LIN {X 0,Y 340.688,Z 497.175,A -85,B 0,C 180,E1 -14276.154,E2 -14276.154} C_VEL
LIN {X 0,Y 340.77,Z 497.165,A -85,B 0,C 180,E1 -14280.333,E2 -14280.333} C_VEL
LIN {X 0,Y 340.804,Z 497.363,A -85,B 0,C 180,E1 -14283.682,E2 -14283.682} C_VEL
LIN {X 0,Y 341.004,Z 498.318,A -85,B 0,C 180,E1 -14283.975,E2 -14283.975} C_VEL
LIN {X 0,Y 342.467,Z 500.978,A -85,B 0,C 180,E1 -14284.442,E2 -14284.442} C_VEL
LIN {X 0,Y 344.948,Z 503.079,A -85,B 0,C 180,E1 -14285.106,E2 -14285.106} C_VEL
LIN {X 0,Y 346.96,Z 506.236,A -85,B 0,C 180,E1 -14285.714,E2 -14285.714} C_VEL
LIN {X 0,Y 349.668,Z 508.622,A -85,B 0,C 180,E1 -14286.488,E2 -14286.488} C_VEL
LIN {X 0,Y 352.115,Z 512,A -85,B 0,C 180,E1 -14287.255,E2 -14287.255} C_VEL
LIN {X 0,Y 355.034,Z 514.578,A -85,B 0,C 180,E1 -14288.144,E2 -14288.144} C_VEL
LIN {X 0,Y 357.879,Z 518.099,A -85,B 0,C 180,E1 -14289.088,E2 -14289.088} C_VEL
LIN {X 0,Y 360.863,Z 520.59,A -85,B 0,C 180,E1 -14290.074,E2 -14290.074} C_VEL
LIN {X 0,Y 363.526,Z 523.831,A -85,B 0,C 180,E1 -14291.039,E2 -14291.039} C_VEL
LIN {X 0,Y 367.234,Z 526.893,A -85,B 0,C 180,E1 -14292.394,E2 -14292.394} C_VEL
LIN {X 0,Y 369.963,Z 530.151,A -85,B 0,C 180,E1 -14293.522,E2 -14293.522} C_VEL
LIN {X 0,Y 373.28,Z 532.615,A -85,B 0,C 180,E1 -14294.922,E2 -14294.922} C_VEL
LIN {X 0,Y 374.392,Z 533.739,A -85,B 0,C 180,E1 -14295.436,E2 -14295.436} C_VEL
LIN {X 0,Y 377.136,Z 536.901,A -85,B 0,C 180,E1 -14296.811,E2 -14296.811} C_VEL
LIN {X 0,Y 380.19,Z 539.057,A -85,B 0,C 180,E1 -14298.441,E2 -14298.441} C_VEL
LIN {X 0,Y 381.738,Z 539.964,A -85,B 0,C 180,E1 -14299.348,E2 -14299.348} C_VEL
LIN {X 0,Y 384.051,Z 542.876,A -85,B 0,C 180,E1 -14301.001,E2 -14301.001} C_VEL
LIN {X 0,Y 386.257,Z 544.769,A -85,B 0,C 180,E1 -14302.826,E2 -14302.826} C_VEL
LIN {X 0,Y 388.334,Z 545.981,A -85,B 0,C 180,E1 -14305.057,E2 -14305.057} C_VEL
LIN {X 0,Y 389.706,Z 546.532,A -85,B 0,C 180,E1 -14307.322,E2 -14307.322} C_VEL
LIN {X 0,Y 390.171,Z 546.851,A -85,B 0,C 180,E1 -14308.968,E2 -14308.968} C_VEL
LIN {X 0,Y 390.171,Z 546.854,A -85,B 0,C 180,E1 -14311.032,E2 -14311.032} C_VEL
LIN {X 0,Y 389.505,Z 546.374,A -85,B 0,C 180,E1 -14313.103,E2 -14313.103} C_VEL
LIN {X 0,Y 388.131,Z 545.895,A -85,B 0,C 180,E1 -14315.197,E2 -14315.197} C_VEL
LIN {X 0,Y 386.111,Z 544.648,A -85,B 0,C 180,E1 -14317.32,E2 -14317.32} C_VEL
LIN {X 0,Y 384.057,Z 542.843,A -85,B 0,C 180,E1 -14318.997,E2 -14318.997} C_VEL
LIN {X 0,Y 381.688,Z 539.897,A -85,B 0,C 180,E1 -14320.684,E2 -14320.684} C_VEL
LIN {X 0,Y 378.266,Z 537.815,A -85,B 0,C 180,E1 -14322.602,E2 -14322.602} C_VEL
LIN {X 0,Y 375.358,Z 535.009,A -85,B 0,C 180,E1 -14324.087,E2 -14324.087} C_VEL
LIN {X 0,Y 373.457,Z 532.737,A -85,B 0,C 180,E1 -14325.002,E2 -14325.002} C_VEL
LIN {X 0,Y 369.922,Z 530.118,A -85,B 0,C 180,E1 -14326.495,E2 -14326.495} C_VEL
LIN {X 0,Y 366.356,Z 526.09,A -85,B 0,C 180,E1 -14327.934,E2 -14327.934} C_VEL
LIN {X 0,Y 362.932,Z 523.255,A -85,B 0,C 180,E1 -14329.176,E2 -14329.176} C_VEL
LIN {X 0,Y 360.249,Z 519.926,A -85,B 0,C 180,E1 -14330.142,E2 -14330.142} C_VEL
LIN {X 0,Y 357.091,Z 517.292,A -85,B 0,C 180,E1 -14331.176,E2 -14331.176} C_VEL
LIN {X 0,Y 354.349,Z 513.844,A -85,B 0,C 180,E1 -14332.076,E2 -14332.076} C_VEL
LIN {X 0,Y 351.341,Z 511.117,A -85,B 0,C 180,E1 -14332.986,E2 -14332.986} C_VEL
LIN {X 0,Y 349.194,Z 508.114,A -85,B 0,C 180,E1 -14333.651,E2 -14333.651} C_VEL
LIN {X 0,Y 346.5,Z 505.693,A -85,B 0,C 180,E1 -14334.417,E2 -14334.417} C_VEL
LIN {X 0,Y 344.728,Z 502.722,A -85,B 0,C 180,E1 -14334.962,E2 -14334.962} C_VEL
LIN {X 0,Y 342.3,Z 500.782,A -85,B 0,C 180,E1 -14335.604,E2 -14335.604} C_VEL
LIN {X 0,Y 340.899,Z 497.904,A -85,B 0,C 180,E1 -14336.105,E2 -14336.105} C_VEL
LIN {X 0,Y 340.809,Z 497.209,A -85,B 0,C 180,E1 -14336.483,E2 -14336.483} C_VEL
LIN {X 0,Y 340.758,Z 497.166,A -85,B 0,C 180,E1 -14339.978,E2 -14339.978} C_VEL
LIN {X 0,Y 340.688,Z 497.175,A -85,B 0,C 180,E1 -14343.846,E2 -14343.846} C_VEL
LIN {X 0,Y 340.7,Z 497.141,A -85,B 0,C 180,E1 -14346.741,E2 -14346.741} C_VEL
LIN {X 0,Y 340.758,Z 497.161,A -85,B 0,C 180,E1 -14350.262,E2 -14350.262} C_VEL
LIN {X 0,Y 340.772,Z 497.12,A -85,B 0,C 180,E1 -14353.795,E2 -14353.795} C_VEL
LIN {X 0,Y 340.755,Z 497.164,A -85,B 0,C 180,E1 -14357.109,E2 -14357.109} C_VEL
LIN {X 0,Y 340.727,Z 497.161,A -85,B 0,C 180,E1 -14360.252,E2 -14360.252} C_VEL
LIN {X 0,Y 340.703,Z 497.158,A -85,B 0,C 180,E1 -14363.559,E2 -14363.559} C_VEL
LIN {X 0,Y 340.688,Z 497.172,A -85,B 0,C 180,E1 -14366.154,E2 -14366.154} C_VEL
LIN {X 0,Y 340.768,Z 497.147,A -85,B 0,C 180,E1 -14370.333,E2 -14370.333} C_VEL
LIN {X 0,Y 340.797,Z 497.156,A -85,B 0,C 180,E1 -14373.02,E2 -14373.02} C_VEL
LIN {X 0,Y 340.753,Z 497.147,A -85,B 0,C 180,E1 -14374.696,E2 -14374.696} C_VEL
LIN {X 0,Y 340.07,Z 497.23,A -85,B 0,C 180,E1 -14375.683,E2 -14375.683} C_VEL
LIN {X 0,Y 337.176,Z 497.602,A -85,B 0,C 180,E1 -14377.288,E2 -14377.288} C_VEL
LIN {X 0,Y 334.755,Z 497.913,A -85,B 0,C 180,E1 -14378.587,E2 -14378.587} C_VEL
LIN {X 0,Y 333.756,Z 498.034,A -85,B 0,C 180,E1 -14379.594,E2 -14379.594} C_VEL
LIN {X 0,Y 333.696,Z 498.037,A -85,B 0,C 180,E1 -14379.935,E2 -14379.935} C_VEL
LIN {X 0,Y 333.738,Z 498.014,A -85,B 0,C 180,E1 -14382.854,E2 -14382.854} C_VEL
LIN {X 0,Y 333.789,Z 498.032,A -85,B 0,C 180,E1 -14386.609,E2 -14386.609} C_VEL
LIN {X 0,Y 333.843,Z 497.997,A -85,B 0,C 180,E1 -14390.305,E2 -14390.305} C_VEL
LIN {X 0,Y 334,Z 498,A -85,B 0,C 180,E1 -14392.748,E2 -14392.748} C_VEL
LIN {X 0,Y 333.807,Z 498.022,A -85,B 0,C 180,E1 -14395.17,E2 -14395.17} C_VEL
LIN {X 0,Y 334.1,Z 497.963,A -85,B 0,C 180,E1 -14397.589,E2 -14397.589} C_VEL
LIN {X 0,Y 334.239,Z 497.962,A -85,B 0,C 180,E1 -14400.001,E2 -14400.001} C_VEL
LIN {X 0,Y 334.1,Z 497.991,A -85,B 0,C 180,E1 -14402.412,E2 -14402.412} C_VEL
LIN {X 0,Y 334.009,Z 497.974,A -85,B 0,C 180,E1 -14406.04,E2 -14406.04} C_VEL
LIN {X 0,Y 333.978,Z 498.003,A -85,B 0,C 180,E1 -14408.502,E2 -14408.502} C_VEL
LIN {X 0,Y 333.784,Z 498.014,A -85,B 0,C 180,E1 -14412.155,E2 -14412.155} C_VEL
LIN {X 0,Y 333.771,Z 498.027,A -85,B 0,C 180,E1 -14415.887,E2 -14415.887} C_VEL
LIN {X 0,Y 333.79,Z 498.023,A -85,B 0,C 180,E1 -14418.656,E2 -14418.656} C_VEL
LIN {X 0,Y 333.651,Z 498.037,A -85,B 0,C 180,E1 -14422.282,E2 -14422.282} C_VEL
LIN {X 0,Y 333.729,Z 498.024,A -85,B 0,C 180,E1 -14426.247,E2 -14426.247} C_VEL
LIN {X 0,Y 333.685,Z 498.039,A -85,B 0,C 180,E1 -14428.975,E2 -14428.975} C_VEL
LIN {X 0,Y 333.639,Z 498.035,A -85,B 0,C 180,E1 -14432.588,E2 -14432.588} C_VEL
LIN {X 0,Y 333.673,Z 498.047,A -85,B 0,C 180,E1 -14436.14,E2 -14436.14} C_VEL
LIN {X 0,Y 333.669,Z 498.045,A -85,B 0,C 180,E1 -14439.19,E2 -14439.19} C_VEL
LIN {X 0,Y 333.663,Z 498.041,A -85,B 0,C 180,E1 -14442.507,E2 -14442.507} C_VEL
LIN {X 0,Y 333.595,Z 498.033,A -85,B 0,C 180,E1 -14445.956,E2 -14445.956} C_VEL
LIN {X 0,Y 333.646,Z 498.051,A -85,B 0,C 180,E1 -14449.316,E2 -14449.316} C_VEL
LIN {X 0,Y 333.679,Z 498.02,A -85,B 0,C 180,E1 -14453.317,E2 -14453.317} C_VEL
LIN {X 0,Y 333.95,Z 499.209,A -85,B 0,C 180,E1 -14453.896,E2 -14453.896} C_VEL
LIN {X 0,Y 336.328,Z 509.72,A -85,B 0,C 180,E1 -14457.448,E2 -14457.448} C_VEL
LIN {X 0,Y 338.327,Z 519.735,A -85,B 0,C 180,E1 -14460.699,E2 -14460.699} C_VEL
LIN {X 0,Y 340.345,Z 524.973,A -85,B 0,C 180,E1 -14461.07,E2 -14461.07} C_VEL
LIN {X 0,Y 342.174,Z 531.358,A -85,B 0,C 180,E1 -14461.387,E2 -14461.387} C_VEL
LIN {X 0,Y 347.112,Z 554.272,A -85,B 0,C 180,E1 -14462.352,E2 -14462.352} C_VEL
LIN {X 0,Y 349.193,Z 565.536,A -85,B 0,C 180,E1 -14462.784,E2 -14462.784} C_VEL
LIN {X 0,Y 346.958,Z 654.163,A -85,B 0,C 180,E1 -14464.626,E2 -14464.626} C_VEL
LIN {X 0,Y 346.331,Z 665.498,A -85,B 0,C 180,E1 -14464.978,E2 -14464.978} C_VEL
LIN {X 0,Y 345.507,Z 676.04,A -85,B 0,C 180,E1 -14465.436,E2 -14465.436} C_VEL
LIN {X 0,Y 344.42,Z 687.192,A -85,B 0,C 180,E1 -14466.075,E2 -14466.075} C_VEL
LIN {X 0,Y 343.36,Z 697.164,A -85,B 0,C 180,E1 -14466.796,E2 -14466.796} C_VEL
LIN {X 0,Y 342.068,Z 706.938,A -85,B 0,C 180,E1 -14467.645,E2 -14467.645} C_VEL
LIN {X 0,Y 340.804,Z 716.811,A -85,B 0,C 180,E1 -14468.688,E2 -14468.688} C_VEL
LIN {X 0,Y 339.314,Z 726.229,A -85,B 0,C 180,E1 -14469.859,E2 -14469.859} C_VEL
LIN {X 0,Y 338.152,Z 733.431,A -85,B 0,C 180,E1 -14470.893,E2 -14470.893} C_VEL
LIN {X 0,Y 336.765,Z 742.226,A -85,B 0,C 180,E1 -14472.386,E2 -14472.386} C_VEL
LIN {X 0,Y 335.551,Z 749.751,A -85,B 0,C 180,E1 -14473.888,E2 -14473.888} C_VEL
LIN {X 0,Y 334.658,Z 756.23,A -85,B 0,C 180,E1 -14475.404,E2 -14475.404} C_VEL
LIN {X 0,Y 333.703,Z 762.773,A -85,B 0,C 180,E1 -14477.225,E2 -14477.225} C_VEL
LIN {X 0,Y 332.883,Z 768.204,A -85,B 0,C 180,E1 -14479.047,E2 -14479.047} C_VEL
LIN {X 0,Y 332.439,Z 772.651,A -85,B 0,C 180,E1 -14480.877,E2 -14480.877} C_VEL
LIN {X 0,Y 332.172,Z 776.198,A -85,B 0,C 180,E1 -14482.707,E2 -14482.707} C_VEL
LIN {X 0,Y 332.004,Z 778.556,A -85,B 0,C 180,E1 -14484.224,E2 -14484.224} C_VEL
LIN {X 0,Y 331.962,Z 780.825,A -85,B 0,C 180,E1 -14486.359,E2 -14486.359} C_VEL
LIN {X 0,Y 331.922,Z 782.114,A -85,B 0,C 180,E1 -14488.787,E2 -14488.787} C_VEL
LIN {X 0,Y 331.969,Z 782.367,A -85,B 0,C 180,E1 -14490,E2 -14490} C_VEL
LIN {X 0,Y 331.913,Z 781.641,A -85,B 0,C 180,E1 -14492.427,E2 -14492.427} C_VEL
LIN {X 0,Y 331.962,Z 780.824,A -85,B 0,C 180,E1 -14493.641,E2 -14493.641} C_VEL
LIN {X 0,Y 332.044,Z 778.139,A -85,B 0,C 180,E1 -14496.075,E2 -14496.075} C_VEL
LIN {X 0,Y 332.241,Z 775.182,A -85,B 0,C 180,E1 -14497.903,E2 -14497.903} C_VEL
LIN {X 0,Y 332.572,Z 771.353,A -85,B 0,C 180,E1 -14499.733,E2 -14499.733} C_VEL
LIN {X 0,Y 333.149,Z 766.589,A -85,B 0,C 180,E1 -14501.561,E2 -14501.561} C_VEL
LIN {X 0,Y 334.095,Z 759.643,A -85,B 0,C 180,E1 -14503.689,E2 -14503.689} C_VEL
LIN {X 0,Y 335.126,Z 752.272,A -85,B 0,C 180,E1 -14505.544,E2 -14505.544} C_VEL
LIN {X 0,Y 336.23,Z 745.35,A -85,B 0,C 180,E1 -14507.015,E2 -14507.015} C_VEL
LIN {X 0,Y 337.581,Z 737.069,A -85,B 0,C 180,E1 -14508.51,E2 -14508.51} C_VEL
LIN {X 0,Y 338.972,Z 728.348,A -85,B 0,C 180,E1 -14509.846,E2 -14509.846} C_VEL
LIN {X 0,Y 340.426,Z 719.291,A -85,B 0,C 180,E1 -14511.02,E2 -14511.02} C_VEL
LIN {X 0,Y 341.744,Z 710.224,A -85,B 0,C 180,E1 -14512.02,E2 -14512.02} C_VEL
LIN {X 0,Y 342.927,Z 700.672,A -85,B 0,C 180,E1 -14512.916,E2 -14512.916} C_VEL
LIN {X 0,Y 344.092,Z 690.413,A -85,B 0,C 180,E1 -14513.71,E2 -14513.71} C_VEL
LIN {X 0,Y 345.127,Z 680.119,A -85,B 0,C 180,E1 -14514.353,E2 -14514.353} C_VEL
LIN {X 0,Y 346.156,Z 668.235,A -85,B 0,C 180,E1 -14514.915,E2 -14514.915} C_VEL
LIN {X 0,Y 346.807,Z 656.819,A -85,B 0,C 180,E1 -14515.306,E2 -14515.306} C_VEL
LIN {X 0,Y 347.758,Z 626.709,A -85,B 0,C 180,E1 -14515.954,E2 -14515.954} C_VEL
LIN {X 0,Y 349.181,Z 565.129,A -85,B 0,C 180,E1 -14517.226,E2 -14517.226} C_VEL
LIN {X 0,Y 344.511,Z 541.355,A -85,B 0,C 180,E1 -14518.171,E2 -14518.171} C_VEL
LIN {X 0,Y 340.705,Z 525.852,A -85,B 0,C 180,E1 -14518.876,E2 -14518.876} C_VEL
LIN {X 0,Y 338.363,Z 519.983,A -85,B 0,C 180,E1 -14519.265,E2 -14519.265} C_VEL
LIN {X 0,Y 337.891,Z 517.596,A -85,B 0,C 180,E1 -14519.946,E2 -14519.946} C_VEL
LIN {X 0,Y 336.034,Z 508.584,A -85,B 0,C 180,E1 -14522.94,E2 -14522.94} C_VEL
LIN {X 0,Y 333.955,Z 499.268,A -85,B 0,C 180,E1 -14526.103,E2 -14526.103} C_VEL
LIN {X 0,Y 333.679,Z 498.035,A -85,B 0,C 180,E1 -14526.683,E2 -14526.683} C_VEL
LIN {X 0,Y 333.646,Z 498.051,A -85,B 0,C 180,E1 -14530.684,E2 -14530.684} C_VEL
LIN {X 0,Y 333.592,Z 498.034,A -85,B 0,C 180,E1 -14534.25,E2 -14534.25} C_VEL
LIN {X 0,Y 333.671,Z 498.038,A -85,B 0,C 180,E1 -14537.622,E2 -14537.622} C_VEL
LIN {X 0,Y 333.674,Z 498.038,A -85,B 0,C 180,E1 -14541.196,E2 -14541.196} C_VEL
LIN {X 0,Y 333.682,Z 498.041,A -85,B 0,C 180,E1 -14545.225,E2 -14545.225} C_VEL
LIN {X 0,Y 333.627,Z 498.046,A -85,B 0,C 180,E1 -14548.221,E2 -14548.221} C_VEL
LIN {X 0,Y 333.685,Z 498.039,A -85,B 0,C 180,E1 -14551.025,E2 -14551.025} C_VEL
LIN {X 0,Y 333.729,Z 498.024,A -85,B 0,C 180,E1 -14553.753,E2 -14553.753} C_VEL
LIN {X 0,Y 333.651,Z 498.037,A -85,B 0,C 180,E1 -14557.718,E2 -14557.718} C_VEL
LIN {X 0,Y 333.788,Z 498.026,A -85,B 0,C 180,E1 -14561.589,E2 -14561.589} C_VEL
LIN {X 0,Y 333.802,Z 498.006,A -85,B 0,C 180,E1 -14565.576,E2 -14565.576} C_VEL
LIN {X 0,Y 333.827,Z 498.021,A -85,B 0,C 180,E1 -14569.077,E2 -14569.077} C_VEL
LIN {X 0,Y 334.007,Z 497.988,A -85,B 0,C 180,E1 -14572.747,E2 -14572.747} C_VEL
LIN {X 0,Y 333.803,Z 498.003,A -85,B 0,C 180,E1 -14575.168,E2 -14575.168} C_VEL
LIN {X 0,Y 334.1,Z 497.991,A -85,B 0,C 180,E1 -14577.588,E2 -14577.588} C_VEL
LIN {X 0,Y 334.239,Z 497.962,A -85,B 0,C 180,E1 -14579.999,E2 -14579.999} C_VEL
LIN {X 0,Y 334.099,Z 497.963,A -85,B 0,C 180,E1 -14582.411,E2 -14582.411} C_VEL
LIN {X 0,Y 333.984,Z 498.001,A -85,B 0,C 180,E1 -14586.66,E2 -14586.66} C_VEL
LIN {X 0,Y 333.843,Z 497.997,A -85,B 0,C 180,E1 -14589.695,E2 -14589.695} C_VEL
LIN {X 0,Y 333.789,Z 498.032,A -85,B 0,C 180,E1 -14593.391,E2 -14593.391} C_VEL
LIN {X 0,Y 333.738,Z 498.014,A -85,B 0,C 180,E1 -14597.146,E2 -14597.146} C_VEL
LIN {X 0,Y 333.729,Z 498.033,A -85,B 0,C 180,E1 -14599.69,E2 -14599.69} C_VEL
LIN {X 0,Y 333.685,Z 498.038,A -85,B 0,C 180,E1 -14602.278,E2 -14602.278} C_VEL
LIN {X 0,Y 333.728,Z 498.035,A -85,B 0,C 180,E1 -14606.246,E2 -14606.246} C_VEL
LIN {X 0,Y 333.704,Z 498.037,A -85,B 0,C 180,E1 -14608.972,E2 -14608.972} C_VEL
LIN {X 0,Y 333.644,Z 498.048,A -85,B 0,C 180,E1 -14612.589,E2 -14612.589} C_VEL
LIN {X 0,Y 333.669,Z 498.032,A -85,B 0,C 180,E1 -14616.139,E2 -14616.139} C_VEL
LIN {X 0,Y 333.675,Z 498.047,A -85,B 0,C 180,E1 -14619.187,E2 -14619.187} C_VEL
LIN {X 0,Y 333.698,Z 498.044,A -85,B 0,C 180,E1 -14622.514,E2 -14622.514} C_VEL
LIN {X 0,Y 333.722,Z 497.999,A -85,B 0,C 180,E1 -14625.977,E2 -14625.977} C_VEL
LIN {X 0,Y 333.695,Z 498.036,A -85,B 0,C 180,E1 -14629.305,E2 -14629.305} C_VEL
LIN {X 0,Y 333.66,Z 498.017,A -85,B 0,C 180,E1 -14633.168,E2 -14633.168} C_VEL
LIN {X 0,Y 333.633,Z 498.053,A -85,B 0,C 180,E1 -14636.792,E2 -14636.792} C_VEL
LIN {X 0,Y 333.697,Z 498.046,A -85,B 0,C 180,E1 -14639.71,E2 -14639.71} C_VEL
LIN {X 0,Y 333.742,Z 498.167,A -85,B 0,C 180,E1 -14642.078,E2 -14642.078} C_VEL
LIN {X 0,Y 333.945,Z 499.111,A -85,B 0,C 180,E1 -14642.42,E2 -14642.42} C_VEL
LIN {X 0,Y 335.52,Z 501.917,A -85,B 0,C 180,E1 -14642.89,E2 -14642.89} C_VEL
LIN {X 0,Y 337.658,Z 503.807,A -85,B 0,C 180,E1 -14643.432,E2 -14643.432} C_VEL
LIN {X 0,Y 339.729,Z 507.005,A -85,B 0,C 180,E1 -14644.011,E2 -14644.011} C_VEL
LIN {X 0,Y 342.228,Z 509.364,A -85,B 0,C 180,E1 -14644.683,E2 -14644.683} C_VEL
LIN {X 0,Y 344.848,Z 512.863,A -85,B 0,C 180,E1 -14645.439,E2 -14645.439} C_VEL
LIN {X 0,Y 347.431,Z 515.31,A -85,B 0,C 180,E1 -14646.165,E2 -14646.165} C_VEL
LIN {X 0,Y 350.369,Z 518.86,A -85,B 0,C 180,E1 -14647.051,E2 -14647.051} C_VEL
LIN {X 0,Y 352.811,Z 521.027,A -85,B 0,C 180,E1 -14647.781,E2 -14647.781} C_VEL
LIN {X 0,Y 356.286,Z 525.015,A -85,B 0,C 180,E1 -14648.905,E2 -14648.905} C_VEL
LIN {X 0,Y 358.943,Z 527.234,A -85,B 0,C 180,E1 -14649.768,E2 -14649.768} C_VEL
LIN {X 0,Y 361.988,Z 530.697,A -85,B 0,C 180,E1 -14650.848,E2 -14650.848} C_VEL
LIN {X 0,Y 365.511,Z 533.647,A -85,B 0,C 180,E1 -14652.126,E2 -14652.126} C_VEL
LIN {X 0,Y 368.669,Z 537.13,A -85,B 0,C 180,E1 -14653.385,E2 -14653.385} C_VEL
LIN {X 0,Y 372.06,Z 539.572,A -85,B 0,C 180,E1 -14654.803,E2 -14654.803} C_VEL
LIN {X 0,Y 375.556,Z 543.504,A -85,B 0,C 180,E1 -14656.485,E2 -14656.485} C_VEL
LIN {X 0,Y 378.664,Z 545.819,A -85,B 0,C 180,E1 -14658.093,E2 -14658.093} C_VEL
LIN {X 0,Y 380.569,Z 546.957,A -85,B 0,C 180,E1 -14659.186,E2 -14659.186} C_VEL
LIN {X 0,Y 383.224,Z 550.114,A -85,B 0,C 180,E1 -14661.059,E2 -14661.059} C_VEL
LIN {X 0,Y 385.511,Z 551.937,A -85,B 0,C 180,E1 -14662.955,E2 -14662.955} C_VEL
LIN {X 0,Y 387.509,Z 553.066,A -85,B 0,C 180,E1 -14665.117,E2 -14665.117} C_VEL
LIN {X 0,Y 388.836,Z 553.579,A -85,B 0,C 180,E1 -14667.316,E2 -14667.316} C_VEL
LIN {X 0,Y 389.306,Z 553.897,A -85,B 0,C 180,E1 -14668.966,E2 -14668.966} C_VEL
LIN {X 0,Y 389.306,Z 553.9,A -85,B 0,C 180,E1 -14671.034,E2 -14671.034} C_VEL
LIN {X 0,Y 388.634,Z 553.424,A -85,B 0,C 180,E1 -14673.11,E2 -14673.11} C_VEL
LIN {X 0,Y 387.253,Z 552.939,A -85,B 0,C 180,E1 -14675.206,E2 -14675.206} C_VEL
LIN {X 0,Y 385.209,Z 551.704,A -85,B 0,C 180,E1 -14677.337,E2 -14677.337} C_VEL
LIN {X 0,Y 383.008,Z 549.847,A -85,B 0,C 180,E1 -14679.114,E2 -14679.114} C_VEL
LIN {X 0,Y 380.501,Z 546.846,A -85,B 0,C 180,E1 -14680.86,E2 -14680.86} C_VEL
LIN {X 0,Y 376.846,Z 544.578,A -85,B 0,C 180,E1 -14682.871,E2 -14682.871} C_VEL
LIN {X 0,Y 373.757,Z 541.622,A -85,B 0,C 180,E1 -14684.397,E2 -14684.397} C_VEL
LIN {X 0,Y 372.058,Z 539.595,A -85,B 0,C 180,E1 -14685.197,E2 -14685.197} C_VEL
LIN {X 0,Y 368.303,Z 536.817,A -85,B 0,C 180,E1 -14686.759,E2 -14686.759} C_VEL
LIN {X 0,Y 364.463,Z 532.646,A -85,B 0,C 180,E1 -14688.272,E2 -14688.272} C_VEL
LIN {X 0,Y 360.971,Z 529.735,A -85,B 0,C 180,E1 -14689.513,E2 -14689.513} C_VEL
LIN {X 0,Y 358.06,Z 526.368,A -85,B 0,C 180,E1 -14690.525,E2 -14690.525} C_VEL
LIN {X 0,Y 354.621,Z 523.361,A -85,B 0,C 180,E1 -14691.624,E2 -14691.624} C_VEL
LIN {X 0,Y 352.152,Z 520.304,A -85,B 0,C 180,E1 -14692.418,E2 -14692.418} C_VEL
LIN {X 0,Y 348.778,Z 517.171,A -85,B 0,C 180,E1 -14693.421,E2 -14693.421} C_VEL
LIN {X 0,Y 346.731,Z 514.452,A -85,B 0,C 180,E1 -14694.045,E2 -14694.045} C_VEL
LIN {X 0,Y 343.594,Z 511.413,A -85,B 0,C 180,E1 -14694.924,E2 -14694.924} C_VEL
LIN {X 0,Y 341.742,Z 508.753,A -85,B 0,C 180,E1 -14695.453,E2 -14695.453} C_VEL
LIN {X 0,Y 339.095,Z 506.226,A -85,B 0,C 180,E1 -14696.158,E2 -14696.158} C_VEL
LIN {X 0,Y 337.294,Z 503.346,A -85,B 0,C 180,E1 -14696.669,E2 -14696.669} C_VEL
LIN {X 0,Y 335.083,Z 501.37,A -85,B 0,C 180,E1 -14697.224,E2 -14697.224} C_VEL
LIN {X 0,Y 333.842,Z 498.648,A -85,B 0,C 180,E1 -14697.681,E2 -14697.681} C_VEL
LIN {X 0,Y 333.71,Z 498.102,A -85,B 0,C 180,E1 -14698.011,E2 -14698.011} C_VEL
LIN {X 0,Y 333.692,Z 498.046,A -85,B 0,C 180,E1 -14700.362,E2 -14700.362} C_VEL
LIN {X 0,Y 333.668,Z 498.043,A -85,B 0,C 180,E1 -14704.658,E2 -14704.658} C_VEL
LIN {X 0,Y 333.65,Z 498.023,A -85,B 0,C 180,E1 -14707.65,E2 -14707.65} C_VEL
LIN {X 0,Y 333.693,Z 498.034,A -85,B 0,C 180,E1 -14710.759,E2 -14710.759} C_VEL
LIN {X 0,Y 333.722,Z 498.002,A -85,B 0,C 180,E1 -14714.274,E2 -14714.274} C_VEL
LIN {X 0,Y 333.7,Z 498.044,A -85,B 0,C 180,E1 -14717.629,E2 -14717.629} C_VEL
LIN {X 0,Y 333.672,Z 498.046,A -85,B 0,C 180,E1 -14721.196,E2 -14721.196} C_VEL
LIN {X 0,Y 333.678,Z 498.04,A -85,B 0,C 180,E1 -14725.226,E2 -14725.226} C_VEL
LIN {X 0,Y 333.636,Z 498.039,A -85,B 0,C 180,E1 -14728.223,E2 -14728.223} C_VEL
LIN {X 0,Y 333.704,Z 498.037,A -85,B 0,C 180,E1 -14731.028,E2 -14731.028} C_VEL
LIN {X 0,Y 333.704,Z 498.025,A -85,B 0,C 180,E1 -14734.701,E2 -14734.701} C_VEL
LIN {X 0,Y 333.712,Z 498.035,A -85,B 0,C 180,E1 -14737.914,E2 -14737.914} C_VEL
LIN {X 0,Y 333.696,Z 498.037,A -85,B 0,C 180,E1 -14739.935,E2 -14739.935} C_VEL
LIN {X 0,Y 333.086,Z 498.113,A -85,B 0,C 180,E1 -14740.942,E2 -14740.942} C_VEL
LIN {X 0,Y 330.261,Z 498.468,A -85,B 0,C 180,E1 -14742.581,E2 -14742.581} C_VEL
LIN {X 0,Y 327.845,Z 498.77,A -85,B 0,C 180,E1 -14743.909,E2 -14743.909} C_VEL
LIN {X 0,Y 326.823,Z 498.897,A -85,B 0,C 180,E1 -14744.937,E2 -14744.937} C_VEL
LIN {X 0,Y 326.75,Z 498.906,A -85,B 0,C 180,E1 -14745.285,E2 -14745.285} C_VEL
LIN {X 0,Y 326.762,Z 498.887,A -85,B 0,C 180,E1 -14748.839,E2 -14748.839} C_VEL
LIN {X 0,Y 326.952,Z 498.875,A -85,B 0,C 180,E1 -14752.59,E2 -14752.59} C_VEL
LIN {X 0,Y 326.773,Z 498.898,A -85,B 0,C 180,E1 -14755.065,E2 -14755.065} C_VEL
LIN {X 0,Y 327.041,Z 498.841,A -85,B 0,C 180,E1 -14757.537,E2 -14757.537} C_VEL
LIN {X 0,Y 327.19,Z 498.84,A -85,B 0,C 180,E1 -14760.001,E2 -14760.001} C_VEL
LIN {X 0,Y 327.041,Z 498.87,A -85,B 0,C 180,E1 -14762.464,E2 -14762.464} C_VEL
LIN {X 0,Y 326.984,Z 498.849,A -85,B 0,C 180,E1 -14766.17,E2 -14766.17} C_VEL
LIN {X 0,Y 326.908,Z 498.886,A -85,B 0,C 180,E1 -14768.656,E2 -14768.656} C_VEL
LIN {X 0,Y 326.727,Z 498.889,A -85,B 0,C 180,E1 -14772.422,E2 -14772.422} C_VEL
LIN {X 0,Y 326.748,Z 498.892,A -85,B 0,C 180,E1 -14774.958,E2 -14774.958} C_VEL
LIN {X 0,Y 326.727,Z 498.9,A -85,B 0,C 180,E1 -14778.839,E2 -14778.839} C_VEL
LIN {X 0,Y 326.597,Z 498.921,A -85,B 0,C 180,E1 -14782.79,E2 -14782.79} C_VEL
LIN {X 0,Y 326.685,Z 498.909,A -85,B 0,C 180,E1 -14785.485,E2 -14785.485} C_VEL
LIN {X 0,Y 326.643,Z 498.92,A -85,B 0,C 180,E1 -14789.661,E2 -14789.661} C_VEL
LIN {X 0,Y 326.603,Z 498.916,A -85,B 0,C 180,E1 -14794.02,E2 -14794.02} C_VEL
LIN {X 0,Y 326.626,Z 498.914,A -85,B 0,C 180,E1 -14797.24,E2 -14797.24} C_VEL
LIN {X 0,Y 326.601,Z 498.929,A -85,B 0,C 180,E1 -14800.208,E2 -14800.208} C_VEL
LIN {X 0,Y 326.576,Z 498.933,A -85,B 0,C 180,E1 -14803.524,E2 -14803.524} C_VEL
LIN {X 0,Y 326.574,Z 498.903,A -85,B 0,C 180,E1 -14807.029,E2 -14807.029} C_VEL
LIN {X 0,Y 326.61,Z 498.892,A -85,B 0,C 180,E1 -14810.774,E2 -14810.774} C_VEL
LIN {X 0,Y 326.631,Z 498.993,A -85,B 0,C 180,E1 -14812.873,E2 -14812.873} C_VEL
LIN {X 0,Y 327.99,Z 504.814,A -85,B 0,C 180,E1 -14815.028,E2 -14815.028} C_VEL
LIN {X 0,Y 329.76,Z 512.88,A -85,B 0,C 180,E1 -14817.805,E2 -14817.805} C_VEL
LIN {X 0,Y 331.026,Z 519.441,A -85,B 0,C 180,E1 -14819.977,E2 -14819.977} C_VEL
LIN {X 0,Y 332.532,Z 523.133,A -85,B 0,C 180,E1 -14820.285,E2 -14820.285} C_VEL
LIN {X 0,Y 335.361,Z 530.523,A -85,B 0,C 180,E1 -14820.736,E2 -14820.736} C_VEL
LIN {X 0,Y 339.896,Z 550.748,A -85,B 0,C 180,E1 -14821.636,E2 -14821.636} C_VEL
LIN {X 0,Y 342.882,Z 566.667,A -85,B 0,C 180,E1 -14822.271,E2 -14822.271} C_VEL
LIN {X 0,Y 340.556,Z 653.972,A -85,B 0,C 180,E1 -14824.114,E2 -14824.114} C_VEL
LIN {X 0,Y 339.903,Z 665.3,A -85,B 0,C 180,E1 -14824.471,E2 -14824.471} C_VEL
LIN {X 0,Y 339.076,Z 675.842,A -85,B 0,C 180,E1 -14824.938,E2 -14824.938} C_VEL
LIN {X 0,Y 337.946,Z 686.994,A -85,B 0,C 180,E1 -14825.587,E2 -14825.587} C_VEL
LIN {X 0,Y 336.826,Z 696.966,A -85,B 0,C 180,E1 -14826.319,E2 -14826.319} C_VEL
LIN {X 0,Y 335.393,Z 707.451,A -85,B 0,C 180,E1 -14827.255,E2 -14827.255} C_VEL
LIN {X 0,Y 334.173,Z 716.612,A -85,B 0,C 180,E1 -14828.243,E2 -14828.243} C_VEL
LIN {X 0,Y 332.648,Z 726.03,A -85,B 0,C 180,E1 -14829.437,E2 -14829.437} C_VEL
LIN {X 0,Y 331.407,Z 733.231,A -85,B 0,C 180,E1 -14830.489,E2 -14830.489} C_VEL
LIN {X 0,Y 329.943,Z 742.027,A -85,B 0,C 180,E1 -14832.01,E2 -14832.01} C_VEL
LIN {X 0,Y 328.695,Z 749.552,A -85,B 0,C 180,E1 -14833.543,E2 -14833.543} C_VEL
LIN {X 0,Y 327.72,Z 756.03,A -85,B 0,C 180,E1 -14835.088,E2 -14835.088} C_VEL
LIN {X 0,Y 326.736,Z 762.573,A -85,B 0,C 180,E1 -14836.947,E2 -14836.947} C_VEL
LIN {X 0,Y 325.867,Z 768.004,A -85,B 0,C 180,E1 -14838.808,E2 -14838.808} C_VEL
LIN {X 0,Y 325.375,Z 772.452,A -85,B 0,C 180,E1 -14840.677,E2 -14840.677} C_VEL
LIN {X 0,Y 325.087,Z 775.999,A -85,B 0,C 180,E1 -14842.547,E2 -14842.547} C_VEL
LIN {X 0,Y 324.906,Z 778.563,A -85,B 0,C 180,E1 -14844.283,E2 -14844.283} C_VEL
LIN {X 0,Y 324.868,Z 780.626,A -85,B 0,C 180,E1 -14846.279,E2 -14846.279} C_VEL
LIN {X 0,Y 324.831,Z 781.916,A -85,B 0,C 180,E1 -14848.76,E2 -14848.76} C_VEL
LIN {X 0,Y 324.873,Z 782.169,A -85,B 0,C 180,E1 -14850,E2 -14850} C_VEL
LIN {X 0,Y 324.832,Z 781.443,A -85,B 0,C 180,E1 -14852.48,E2 -14852.48} C_VEL
LIN {X 0,Y 324.868,Z 780.626,A -85,B 0,C 180,E1 -14853.721,E2 -14853.721} C_VEL
LIN {X 0,Y 324.96,Z 777.94,A -85,B 0,C 180,E1 -14856.208,E2 -14856.208} C_VEL
LIN {X 0,Y 325.176,Z 774.983,A -85,B 0,C 180,E1 -14858.076,E2 -14858.076} C_VEL
LIN {X 0,Y 325.522,Z 771.153,A -85,B 0,C 180,E1 -14859.946,E2 -14859.946} C_VEL
LIN {X 0,Y 326.142,Z 766.39,A -85,B 0,C 180,E1 -14861.812,E2 -14861.812} C_VEL
LIN {X 0,Y 327.15,Z 759.444,A -85,B 0,C 180,E1 -14863.985,E2 -14863.985} C_VEL
LIN {X 0,Y 328.217,Z 752.247,A -85,B 0,C 180,E1 -14865.839,E2 -14865.839} C_VEL
LIN {X 0,Y 329.408,Z 745.151,A -85,B 0,C 180,E1 -14867.379,E2 -14867.379} C_VEL
LIN {X 0,Y 330.8,Z 736.87,A -85,B 0,C 180,E1 -14868.904,E2 -14868.904} C_VEL
LIN {X 0,Y 332.235,Z 728.148,A -85,B 0,C 180,E1 -14870.266,E2 -14870.266} C_VEL
LIN {X 0,Y 333.792,Z 719.093,A -85,B 0,C 180,E1 -14871.458,E2 -14871.458} C_VEL
LIN {X 0,Y 335.015,Z 711.014,A -85,B 0,C 180,E1 -14872.377,E2 -14872.377} C_VEL
LIN {X 0,Y 336.373,Z 700.473,A -85,B 0,C 180,E1 -14873.389,E2 -14873.389} C_VEL
LIN {X 0,Y 337.583,Z 690.214,A -85,B 0,C 180,E1 -14874.196,E2 -14874.196} C_VEL
LIN {X 0,Y 338.68,Z 679.921,A -85,B 0,C 180,E1 -14874.847,E2 -14874.847} C_VEL
LIN {X 0,Y 339.746,Z 668.037,A -85,B 0,C 180,E1 -14875.418,E2 -14875.418} C_VEL
LIN {X 0,Y 340.414,Z 656.622,A -85,B 0,C 180,E1 -14875.816,E2 -14875.816} C_VEL
LIN {X 0,Y 341.398,Z 626.512,A -85,B 0,C 180,E1 -14876.475,E2 -14876.475} C_VEL
LIN {X 0,Y 342.773,Z 565.761,A -85,B 0,C 180,E1 -14877.759,E2 -14877.759} C_VEL
LIN {X 0,Y 338.456,Z 543.649,A -85,B 0,C 180,E1 -14878.663,E2 -14878.663} C_VEL
LIN {X 0,Y 334.803,Z 528.674,A -85,B 0,C 180,E1 -14879.362,E2 -14879.362} C_VEL
LIN {X 0,Y 331.154,Z 519.8,A -85,B 0,C 180,E1 -14879.961,E2 -14879.961} C_VEL
LIN {X 0,Y 330.655,Z 517.36,A -85,B 0,C 180,E1 -14880.671,E2 -14880.671} C_VEL
LIN {X 0,Y 328.824,Z 508.344,A -85,B 0,C 180,E1 -14883.758,E2 -14883.758} C_VEL
LIN {X 0,Y 326.652,Z 499.146,A -85,B 0,C 180,E1 -14887.043,E2 -14887.043} C_VEL
LIN {X 0,Y 326.626,Z 498.908,A -85,B 0,C 180,E1 -14887.238,E2 -14887.238} C_VEL
LIN {X 0,Y 326.577,Z 498.928,A -85,B 0,C 180,E1 -14891.13,E2 -14891.13} C_VEL
LIN {X 0,Y 326.528,Z 498.92,A -85,B 0,C 180,E1 -14894.742,E2 -14894.742} C_VEL
LIN {X 0,Y 326.595,Z 498.918,A -85,B 0,C 180,E1 -14898.157,E2 -14898.157} C_VEL
LIN {X 0,Y 326.64,Z 498.912,A -85,B 0,C 180,E1 -14901.393,E2 -14901.393} C_VEL
LIN {X 0,Y 326.616,Z 498.926,A -85,B 0,C 180,E1 -14904.85,E2 -14904.85} C_VEL
LIN {X 0,Y 326.603,Z 498.911,A -85,B 0,C 180,E1 -14907.455,E2 -14907.455} C_VEL
LIN {X 0,Y 326.643,Z 498.92,A -85,B 0,C 180,E1 -14910.339,E2 -14910.339} C_VEL
LIN {X 0,Y 326.685,Z 498.909,A -85,B 0,C 180,E1 -14914.515,E2 -14914.515} C_VEL
LIN {X 0,Y 326.613,Z 498.906,A -85,B 0,C 180,E1 -14918.542,E2 -14918.542} C_VEL
LIN {X 0,Y 326.739,Z 498.899,A -85,B 0,C 180,E1 -14921.177,E2 -14921.177} C_VEL
LIN {X 0,Y 326.757,Z 498.885,A -85,B 0,C 180,E1 -14925.433,E2 -14925.433} C_VEL
LIN {X 0,Y 326.763,Z 498.899,A -85,B 0,C 180,E1 -14928.838,E2 -14928.838} C_VEL
LIN {X 0,Y 326.961,Z 498.868,A -85,B 0,C 180,E1 -14932.589,E2 -14932.589} C_VEL
LIN {X 0,Y 326.77,Z 498.878,A -85,B 0,C 180,E1 -14935.064,E2 -14935.064} C_VEL
LIN {X 0,Y 327.041,Z 498.87,A -85,B 0,C 180,E1 -14937.536,E2 -14937.536} C_VEL
LIN {X 0,Y 327.19,Z 498.84,A -85,B 0,C 180,E1 -14939.999,E2 -14939.999} C_VEL
LIN {X 0,Y 327.04,Z 498.841,A -85,B 0,C 180,E1 -14942.463,E2 -14942.463} C_VEL
LIN {X 0,Y 326.951,Z 498.876,A -85,B 0,C 180,E1 -14946.652,E2 -14946.652} C_VEL
LIN {X 0,Y 326.798,Z 498.874,A -85,B 0,C 180,E1 -14949.906,E2 -14949.906} C_VEL
LIN {X 0,Y 326.751,Z 498.911,A -85,B 0,C 180,E1 -14953.685,E2 -14953.685} C_VEL
LIN {X 0,Y 326.69,Z 498.891,A -85,B 0,C 180,E1 -14957.528,E2 -14957.528} C_VEL
LIN {X 0,Y 326.656,Z 498.92,A -85,B 0,C 180,E1 -14960.135,E2 -14960.135} C_VEL
LIN {X 0,Y 326.644,Z 498.898,A -85,B 0,C 180,E1 -14964.129,E2 -14964.129} C_VEL
LIN {X 0,Y 326.678,Z 498.915,A -85,B 0,C 180,E1 -14966.857,E2 -14966.857} C_VEL
LIN {X 0,Y 326.634,Z 498.902,A -85,B 0,C 180,E1 -14970.612,E2 -14970.612} C_VEL
LIN {X 0,Y 326.601,Z 498.925,A -85,B 0,C 180,E1 -14974.019,E2 -14974.019} C_VEL
LIN {X 0,Y 326.621,Z 498.917,A -85,B 0,C 180,E1 -14977.239,E2 -14977.239} C_VEL
LIN {X 0,Y 326.628,Z 498.912,A -85,B 0,C 180,E1 -14980.203,E2 -14980.203} C_VEL
LIN {X 0,Y 326.652,Z 498.921,A -85,B 0,C 180,E1 -14983.51,E2 -14983.51} C_VEL
LIN {X 0,Y 326.643,Z 498.875,A -85,B 0,C 180,E1 -14987.014,E2 -14987.014} C_VEL
LIN {X 0,Y 326.639,Z 498.923,A -85,B 0,C 180,E1 -14990.766,E2 -14990.766} C_VEL
LIN {X 0,Y 326.606,Z 498.903,A -85,B 0,C 180,E1 -14994.481,E2 -14994.481} C_VEL
LIN {X 0,Y 326.604,Z 498.929,A -85,B 0,C 180,E1 -14997.456,E2 -14997.456} C_VEL
LIN {X 0,Y 326.687,Z 499.152,A -85,B 0,C 180,E1 -15000.698,E2 -15000.698} C_VEL
LIN {X 0,Y 326.937,Z 500.179,A -85,B 0,C 180,E1 -15000.991,E2 -15000.991} C_VEL
LIN {X 0,Y 328.443,Z 502.79,A -85,B 0,C 180,E1 -15001.399,E2 -15001.399} C_VEL
LIN {X 0,Y 330.481,Z 504.645,A -85,B 0,C 180,E1 -15001.895,E2 -15001.895} C_VEL
LIN {X 0,Y 332.627,Z 507.889,A -85,B 0,C 180,E1 -15002.458,E2 -15002.458} C_VEL
LIN {X 0,Y 334.792,Z 510.055,A -85,B 0,C 180,E1 -15003.008,E2 -15003.008} C_VEL
LIN {X 0,Y 337.389,Z 513.515,A -85,B 0,C 180,E1 -15003.709,E2 -15003.709} C_VEL
LIN {X 0,Y 339.667,Z 515.771,A -85,B 0,C 180,E1 -15004.305,E2 -15004.305} C_VEL
LIN {X 0,Y 342.741,Z 519.475,A -85,B 0,C 180,E1 -15005.161,E2 -15005.161} C_VEL
LIN {X 0,Y 344.825,Z 521.462,A -85,B 0,C 180,E1 -15005.745,E2 -15005.745} C_VEL
LIN {X 0,Y 348.183,Z 525.325,A -85,B 0,C 180,E1 -15006.73,E2 -15006.73} C_VEL
LIN {X 0,Y 350.587,Z 527.525,A -85,B 0,C 180,E1 -15007.443,E2 -15007.443} C_VEL
LIN {X 0,Y 354.159,Z 531.452,A -85,B 0,C 180,E1 -15008.566,E2 -15008.566} C_VEL
LIN {X 0,Y 356.816,Z 533.689,A -85,B 0,C 180,E1 -15009.413,E2 -15009.413} C_VEL
LIN {X 0,Y 360.134,Z 537.29,A -85,B 0,C 180,E1 -15010.551,E2 -15010.551} C_VEL
LIN {X 0,Y 363.674,Z 540.237,A -85,B 0,C 180,E1 -15011.809,E2 -15011.809} C_VEL
LIN {X 0,Y 367.005,Z 543.812,A -85,B 0,C 180,E1 -15013.116,E2 -15013.116} C_VEL
LIN {X 0,Y 371.123,Z 546.975,A -85,B 0,C 180,E1 -15014.818,E2 -15014.818} C_VEL
LIN {X 0,Y 374.364,Z 550.486,A -85,B 0,C 180,E1 -15016.353,E2 -15016.353} C_VEL
LIN {X 0,Y 377.541,Z 552.79,A -85,B 0,C 180,E1 -15017.981,E2 -15017.981} C_VEL
LIN {X 0,Y 379.321,Z 553.833,A -85,B 0,C 180,E1 -15018.98,E2 -15018.98} C_VEL
LIN {X 0,Y 382.198,Z 557.115,A -85,B 0,C 180,E1 -15020.957,E2 -15020.957} C_VEL
LIN {X 0,Y 384.616,Z 558.989,A -85,B 0,C 180,E1 -15022.939,E2 -15022.939} C_VEL
LIN {X 0,Y 386.628,Z 560.112,A -85,B 0,C 180,E1 -15025.106,E2 -15025.106} C_VEL
LIN {X 0,Y 387.964,Z 560.626,A -85,B 0,C 180,E1 -15027.31,E2 -15027.31} C_VEL
LIN {X 0,Y 388.44,Z 560.943,A -85,B 0,C 180,E1 -15028.963,E2 -15028.963} C_VEL
LIN {X 0,Y 388.44,Z 560.946,A -85,B 0,C 180,E1 -15031.037,E2 -15031.037} C_VEL
LIN {X 0,Y 387.763,Z 560.46,A -85,B 0,C 180,E1 -15033.117,E2 -15033.117} C_VEL
LIN {X 0,Y 386.372,Z 559.988,A -85,B 0,C 180,E1 -15035.218,E2 -15035.218} C_VEL
LIN {X 0,Y 384.303,Z 558.763,A -85,B 0,C 180,E1 -15037.355,E2 -15037.355} C_VEL
LIN {X 0,Y 381.96,Z 556.847,A -85,B 0,C 180,E1 -15039.232,E2 -15039.232} C_VEL
LIN {X 0,Y 379.334,Z 553.823,A -85,B 0,C 180,E1 -15041.013,E2 -15041.013} C_VEL
LIN {X 0,Y 375.57,Z 551.47,A -85,B 0,C 180,E1 -15043.044,E2 -15043.044} C_VEL
LIN {X 0,Y 372.288,Z 548.381,A -85,B 0,C 180,E1 -15044.649,E2 -15044.649} C_VEL
LIN {X 0,Y 370.533,Z 546.377,A -85,B 0,C 180,E1 -15045.449,E2 -15045.449} C_VEL
LIN {X 0,Y 366.629,Z 543.477,A -85,B 0,C 180,E1 -15047.032,E2 -15047.032} C_VEL
LIN {X 0,Y 362.627,Z 539.274,A -85,B 0,C 180,E1 -15048.576,E2 -15048.576} C_VEL
LIN {X 0,Y 358.846,Z 536.082,A -85,B 0,C 180,E1 -15049.888,E2 -15049.888} C_VEL
LIN {X 0,Y 356.16,Z 533.002,A -85,B 0,C 180,E1 -15050.804,E2 -15050.804} C_VEL
LIN {X 0,Y 352.347,Z 529.653,A -85,B 0,C 180,E1 -15052.009,E2 -15052.009} C_VEL
LIN {X 0,Y 349.507,Z 526.431,A -85,B 0,C 180,E1 -15052.888,E2 -15052.888} C_VEL
LIN {X 0,Y 345.84,Z 522.802,A -85,B 0,C 180,E1 -15053.96,E2 -15053.96} C_VEL
LIN {X 0,Y 343.817,Z 520.408,A -85,B 0,C 180,E1 -15054.541,E2 -15054.541} C_VEL
LIN {X 0,Y 340.489,Z 516.956,A -85,B 0,C 180,E1 -15055.458,E2 -15055.458} C_VEL
LIN {X 0,Y 338.775,Z 514.735,A -85,B 0,C 180,E1 -15055.936,E2 -15055.936} C_VEL
LIN {X 0,Y 335.738,Z 511.499,A -85,B 0,C 180,E1 -15056.738,E2 -15056.738} C_VEL
LIN {X 0,Y 334.023,Z 509.165,A -85,B 0,C 180,E1 -15057.19,E2 -15057.19} C_VEL
LIN {X 0,Y 331.696,Z 506.661,A -85,B 0,C 180,E1 -15057.783,E2 -15057.783} C_VEL
LIN {X 0,Y 330.012,Z 504.131,A -85,B 0,C 180,E1 -15058.222,E2 -15058.222} C_VEL
LIN {X 0,Y 327.841,Z 502.023,A -85,B 0,C 180,E1 -15058.748,E2 -15058.748} C_VEL
LIN {X 0,Y 326.77,Z 499.595,A -85,B 0,C 180,E1 -15059.131,E2 -15059.131} C_VEL
LIN {X 0,Y 326.653,Z 498.992,A -85,B 0,C 180,E1 -15059.482,E2 -15059.482} C_VEL
LIN {X 0,Y 326.613,Z 498.928,A -85,B 0,C 180,E1 -15062.946,E2 -15062.946} C_VEL
LIN {X 0,Y 326.606,Z 498.903,A -85,B 0,C 180,E1 -15065.519,E2 -15065.519} C_VEL
LIN {X 0,Y 326.639,Z 498.923,A -85,B 0,C 180,E1 -15069.234,E2 -15069.234} C_VEL
LIN {X 0,Y 326.643,Z 498.875,A -85,B 0,C 180,E1 -15072.986,E2 -15072.986} C_VEL
LIN {X 0,Y 326.652,Z 498.921,A -85,B 0,C 180,E1 -15076.49,E2 -15076.49} C_VEL
LIN {X 0,Y 326.628,Z 498.912,A -85,B 0,C 180,E1 -15079.797,E2 -15079.797} C_VEL
LIN {X 0,Y 326.623,Z 498.916,A -85,B 0,C 180,E1 -15082.953,E2 -15082.953} C_VEL
LIN {X 0,Y 326.615,Z 498.924,A -85,B 0,C 180,E1 -15087.052,E2 -15087.052} C_VEL
LIN {X 0,Y 326.654,Z 498.904,A -85,B 0,C 180,E1 -15090.341,E2 -15090.341} C_VEL
LIN {X 0,Y 326.682,Z 498.901,A -85,B 0,C 180,E1 -15094.516,E2 -15094.516} C_VEL
LIN {X 0,Y 326.638,Z 498.923,A -85,B 0,C 180,E1 -15098.545,E2 -15098.545} C_VEL
LIN {X 0,Y 326.737,Z 498.897,A -85,B 0,C 180,E1 -15101.178,E2 -15101.178} C_VEL
LIN {X 0,Y 326.75,Z 498.906,A -85,B 0,C 180,E1 -15105.285,E2 -15105.285} C_VEL
LIN {X 0,Y 326.1,Z 498.992,A -85,B 0,C 180,E1 -15106.314,E2 -15106.314} C_VEL
LIN {X 0,Y 323.233,Z 499.337,A -85,B 0,C 180,E1 -15107.988,E2 -15107.988} C_VEL
LIN {X 0,Y 320.824,Z 499.623,A -85,B 0,C 180,E1 -15109.345,E2 -15109.345} C_VEL
LIN {X 0,Y 319.839,Z 499.741,A -85,B 0,C 180,E1 -15110.396,E2 -15110.396} C_VEL
LIN {X 0,Y 319.786,Z 499.749,A -85,B 0,C 180,E1 -15110.752,E2 -15110.752} C_VEL
LIN {X 0,Y 319.939,Z 499.753,A -85,B 0,C 180,E1 -15113.695,E2 -15113.695} C_VEL
LIN {X 0,Y 319.985,Z 499.72,A -85,B 0,C 180,E1 -15117.483,E2 -15117.483} C_VEL
LIN {X 0,Y 320.142,Z 499.718,A -85,B 0,C 180,E1 -15120.001,E2 -15120.001} C_VEL
LIN {X 0,Y 319.985,Z 499.748,A -85,B 0,C 180,E1 -15122.518,E2 -15122.518} C_VEL
LIN {X 0,Y 319.939,Z 499.726,A -85,B 0,C 180,E1 -15126.306,E2 -15126.306} C_VEL
LIN {X 0,Y 319.836,Z 499.769,A -85,B 0,C 180,E1 -15128.849,E2 -15128.849} C_VEL
LIN {X 0,Y 319.674,Z 499.763,A -85,B 0,C 180,E1 -15132.701,E2 -15132.701} C_VEL
LIN {X 0,Y 319.694,Z 499.776,A -85,B 0,C 180,E1 -15135.296,E2 -15135.296} C_VEL
LIN {X 0,Y 319.646,Z 499.779,A -85,B 0,C 180,E1 -15139.257,E2 -15139.257} C_VEL
LIN {X 0,Y 319.555,Z 499.803,A -85,B 0,C 180,E1 -15143.321,E2 -15143.321} C_VEL
LIN {X 0,Y 319.613,Z 499.783,A -85,B 0,C 180,E1 -15146.09,E2 -15146.09} C_VEL
LIN {X 0,Y 319.575,Z 499.795,A -85,B 0,C 180,E1 -15148.936,E2 -15148.936} C_VEL
LIN {X 0,Y 319.526,Z 499.799,A -85,B 0,C 180,E1 -15151.863,E2 -15151.863} C_VEL
LIN {X 0,Y 319.577,Z 499.802,A -85,B 0,C 180,E1 -15155.544,E2 -15155.544} C_VEL
LIN {X 0,Y 319.579,Z 499.789,A -85,B 0,C 180,E1 -15158.008,E2 -15158.008} C_VEL
LIN {X 0,Y 319.566,Z 499.796,A -85,B 0,C 180,E1 -15161.607,E2 -15161.607} C_VEL
LIN {X 0,Y 319.489,Z 499.798,A -85,B 0,C 180,E1 -15165.259,E2 -15165.259} C_VEL
LIN {X 0,Y 319.527,Z 499.802,A -85,B 0,C 180,E1 -15168.713,E2 -15168.713} C_VEL
LIN {X 0,Y 319.582,Z 499.952,A -85,B 0,C 180,E1 -15172.344,E2 -15172.344} C_VEL
LIN {X 0,Y 321.115,Z 506.435,A -85,B 0,C 180,E1 -15174.765,E2 -15174.765} C_VEL
LIN {X 0,Y 323.098,Z 515.601,A -85,B 0,C 180,E1 -15178.031,E2 -15178.031} C_VEL
LIN {X 0,Y 323.884,Z 519.442,A -85,B 0,C 180,E1 -15179.281,E2 -15179.281} C_VEL
LIN {X 0,Y 329.295,Z 532.437,A -85,B 0,C 180,E1 -15180.194,E2 -15180.194} C_VEL
LIN {X 0,Y 333.992,Z 553.733,A -85,B 0,C 180,E1 -15181.164,E2 -15181.164} C_VEL
LIN {X 0,Y 336.579,Z 567.853,A -85,B 0,C 180,E1 -15181.739,E2 -15181.739} C_VEL
LIN {X 0,Y 334.196,Z 653.782,A -85,B 0,C 180,E1 -15183.583,E2 -15183.583} C_VEL
LIN {X 0,Y 333.513,Z 665.102,A -85,B 0,C 180,E1 -15183.946,E2 -15183.946} C_VEL
LIN {X 0,Y 332.665,Z 675.644,A -85,B 0,C 180,E1 -15184.421,E2 -15184.421} C_VEL
LIN {X 0,Y 331.472,Z 686.795,A -85,B 0,C 180,E1 -15185.078,E2 -15185.078} C_VEL
LIN {X 0,Y 330.313,Z 696.767,A -85,B 0,C 180,E1 -15185.822,E2 -15185.822} C_VEL
LIN {X 0,Y 329.027,Z 706.011,A -85,B 0,C 180,E1 -15186.648,E2 -15186.648} C_VEL
LIN {X 0,Y 327.557,Z 716.413,A -85,B 0,C 180,E1 -15187.781,E2 -15187.781} C_VEL
LIN {X 0,Y 325.999,Z 725.832,A -85,B 0,C 180,E1 -15188.998,E2 -15188.998} C_VEL
LIN {X 0,Y 324.362,Z 734.851,A -85,B 0,C 180,E1 -15190.377,E2 -15190.377} C_VEL
LIN {X 0,Y 323.152,Z 741.827,A -85,B 0,C 180,E1 -15191.618,E2 -15191.618} C_VEL
LIN {X 0,Y 321.845,Z 749.352,A -85,B 0,C 180,E1 -15193.182,E2 -15193.182} C_VEL
LIN {X 0,Y 320.775,Z 755.829,A -85,B 0,C 180,E1 -15194.757,E2 -15194.757} C_VEL
LIN {X 0,Y 319.769,Z 762.374,A -85,B 0,C 180,E1 -15196.658,E2 -15196.658} C_VEL
LIN {X 0,Y 318.855,Z 767.805,A -85,B 0,C 180,E1 -15198.559,E2 -15198.559} C_VEL
LIN {X 0,Y 318.32,Z 772.252,A -85,B 0,C 180,E1 -15200.469,E2 -15200.469} C_VEL
LIN {X 0,Y 318.012,Z 775.8,A -85,B 0,C 180,E1 -15202.38,E2 -15202.38} C_VEL
LIN {X 0,Y 317.821,Z 778.545,A -85,B 0,C 180,E1 -15204.322,E2 -15204.322} C_VEL
LIN {X 0,Y 317.778,Z 780.428,A -85,B 0,C 180,E1 -15206.196,E2 -15206.196} C_VEL
LIN {X 0,Y 317.742,Z 781.719,A -85,B 0,C 180,E1 -15208.733,E2 -15208.733} C_VEL
LIN {X 0,Y 317.781,Z 781.972,A -85,B 0,C 180,E1 -15210,E2 -15210} C_VEL
LIN {X 0,Y 317.753,Z 781.245,A -85,B 0,C 180,E1 -15212.535,E2 -15212.535} C_VEL
LIN {X 0,Y 317.778,Z 780.428,A -85,B 0,C 180,E1 -15213.804,E2 -15213.804} C_VEL
LIN {X 0,Y 317.885,Z 777.742,A -85,B 0,C 180,E1 -15216.346,E2 -15216.346} C_VEL
LIN {X 0,Y 318.106,Z 774.783,A -85,B 0,C 180,E1 -15218.256,E2 -15218.256} C_VEL
LIN {X 0,Y 318.491,Z 770.954,A -85,B 0,C 180,E1 -15220.168,E2 -15220.168} C_VEL
LIN {X 0,Y 319.148,Z 766.19,A -85,B 0,C 180,E1 -15222.075,E2 -15222.075} C_VEL
LIN {X 0,Y 320.229,Z 759.244,A -85,B 0,C 180,E1 -15224.294,E2 -15224.294} C_VEL
LIN {X 0,Y 321.336,Z 752.029,A -85,B 0,C 180,E1 -15226.191,E2 -15226.191} C_VEL
LIN {X 0,Y 322.582,Z 744.951,A -85,B 0,C 180,E1 -15227.759,E2 -15227.759} C_VEL
LIN {X 0,Y 324.043,Z 736.67,A -85,B 0,C 180,E1 -15229.314,E2 -15229.314} C_VEL
LIN {X 0,Y 325.575,Z 727.949,A -85,B 0,C 180,E1 -15230.7,E2 -15230.7} C_VEL
LIN {X 0,Y 327.186,Z 718.895,A -85,B 0,C 180,E1 -15231.914,E2 -15231.914} C_VEL
LIN {X 0,Y 328.54,Z 709.911,A -85,B 0,C 180,E1 -15232.945,E2 -15232.945} C_VEL
LIN {X 0,Y 329.856,Z 700.275,A -85,B 0,C 180,E1 -15233.879,E2 -15233.879} C_VEL
LIN {X 0,Y 331.092,Z 690.015,A -85,B 0,C 180,E1 -15234.702,E2 -15234.702} C_VEL
LIN {X 0,Y 332.392,Z 678.364,A -85,B 0,C 180,E1 -15235.434,E2 -15235.434} C_VEL
LIN {X 0,Y 333.342,Z 667.839,A -85,B 0,C 180,E1 -15235.943,E2 -15235.943} C_VEL
LIN {X 0,Y 334.052,Z 656.424,A -85,B 0,C 180,E1 -15236.345,E2 -15236.345} C_VEL
LIN {X 0,Y 335.047,Z 626.313,A -85,B 0,C 180,E1 -15237.017,E2 -15237.017} C_VEL
LIN {X 0,Y 336.492,Z 566.815,A -85,B 0,C 180,E1 -15238.294,E2 -15238.294} C_VEL
LIN {X 0,Y 331.659,Z 542.395,A -85,B 0,C 180,E1 -15239.332,E2 -15239.332} C_VEL
LIN {X 0,Y 328.971,Z 531.487,A -85,B 0,C 180,E1 -15239.861,E2 -15239.861} C_VEL
LIN {X 0,Y 323.883,Z 519.456,A -85,B 0,C 180,E1 -15240.717,E2 -15240.717} C_VEL
LIN {X 0,Y 323.112,Z 515.585,A -85,B 0,C 180,E1 -15241.973,E2 -15241.973} C_VEL
LIN {X 0,Y 321.155,Z 506.444,A -85,B 0,C 180,E1 -15245.23,E2 -15245.23} C_VEL
LIN {X 0,Y 319.564,Z 499.865,A -85,B 0,C 180,E1 -15247.718,E2 -15247.718} C_VEL
LIN {X 0,Y 319.527,Z 499.802,A -85,B 0,C 180,E1 -15251.287,E2 -15251.287} C_VEL
LIN {X 0,Y 319.489,Z 499.796,A -85,B 0,C 180,E1 -15254.741,E2 -15254.741} C_VEL
LIN {X 0,Y 319.566,Z 499.794,A -85,B 0,C 180,E1 -15258.393,E2 -15258.393} C_VEL
LIN {X 0,Y 319.579,Z 499.789,A -85,B 0,C 180,E1 -15262.342,E2 -15262.342} C_VEL
LIN {X 0,Y 319.557,Z 499.801,A -85,B 0,C 180,E1 -15265.122,E2 -15265.122} C_VEL
LIN {X 0,Y 319.562,Z 499.801,A -85,B 0,C 180,E1 -15269.058,E2 -15269.058} C_VEL
LIN {X 0,Y 319.6,Z 499.778,A -85,B 0,C 180,E1 -15272.497,E2 -15272.497} C_VEL
LIN {X 0,Y 319.598,Z 499.797,A -85,B 0,C 180,E1 -15275.303,E2 -15275.303} C_VEL
LIN {X 0,Y 319.596,Z 499.775,A -85,B 0,C 180,E1 -15279.399,E2 -15279.399} C_VEL
LIN {X 0,Y 319.652,Z 499.791,A -85,B 0,C 180,E1 -15282.072,E2 -15282.072} C_VEL
LIN {X 0,Y 319.726,Z 499.755,A -85,B 0,C 180,E1 -15286.007,E2 -15286.007} C_VEL
LIN {X 0,Y 319.75,Z 499.781,A -85,B 0,C 180,E1 -15289.872,E2 -15289.872} C_VEL
LIN {X 0,Y 319.919,Z 499.748,A -85,B 0,C 180,E1 -15292.425,E2 -15292.425} C_VEL
LIN {X 0,Y 319.739,Z 499.752,A -85,B 0,C 180,E1 -15294.955,E2 -15294.955} C_VEL
LIN {X 0,Y 319.984,Z 499.748,A -85,B 0,C 180,E1 -15297.482,E2 -15297.482} C_VEL
LIN {X 0,Y 320.142,Z 499.718,A -85,B 0,C 180,E1 -15299.999,E2 -15299.999} C_VEL
LIN {X 0,Y 319.984,Z 499.72,A -85,B 0,C 180,E1 -15302.517,E2 -15302.517} C_VEL
LIN {X 0,Y 319.913,Z 499.753,A -85,B 0,C 180,E1 -15306.64,E2 -15306.64} C_VEL
LIN {X 0,Y 319.745,Z 499.752,A -85,B 0,C 180,E1 -15310.127,E2 -15310.127} C_VEL
LIN {X 0,Y 319.723,Z 499.781,A -85,B 0,C 180,E1 -15314.724,E2 -15314.724} C_VEL
LIN {X 0,Y 319.681,Z 499.776,A -85,B 0,C 180,E1 -15319.037,E2 -15319.037} C_VEL
LIN {X 0,Y 319.562,Z 499.785,A -85,B 0,C 180,E1 -15323.319,E2 -15323.319} C_VEL
LIN {X 0,Y 319.627,Z 499.787,A -85,B 0,C 180,E1 -15326.088,E2 -15326.088} C_VEL
LIN {X 0,Y 319.583,Z 499.795,A -85,B 0,C 180,E1 -15328.933,E2 -15328.933} C_VEL
LIN {X 0,Y 319.531,Z 499.796,A -85,B 0,C 180,E1 -15331.861,E2 -15331.861} C_VEL
LIN {X 0,Y 319.572,Z 499.788,A -85,B 0,C 180,E1 -15335.543,E2 -15335.543} C_VEL
LIN {X 0,Y 319.591,Z 499.801,A -85,B 0,C 180,E1 -15338.005,E2 -15338.005} C_VEL
LIN {X 0,Y 319.595,Z 499.789,A -85,B 0,C 180,E1 -15341.613,E2 -15341.613} C_VEL
LIN {X 0,Y 319.639,Z 499.762,A -85,B 0,C 180,E1 -15345.285,E2 -15345.285} C_VEL
LIN {X 0,Y 319.576,Z 499.775,A -85,B 0,C 180,E1 -15348.72,E2 -15348.72} C_VEL
LIN {X 0,Y 319.577,Z 499.775,A -85,B 0,C 180,E1 -15352.343,E2 -15352.343} C_VEL
LIN {X 0,Y 319.554,Z 499.793,A -85,B 0,C 180,E1 -15355.124,E2 -15355.124} C_VEL
LIN {X 0,Y 319.583,Z 499.872,A -85,B 0,C 180,E1 -15359.216,E2 -15359.216} C_VEL
LIN {X 0,Y 319.744,Z 500.64,A -85,B 0,C 180,E1 -15359.564,E2 -15359.564} C_VEL
LIN {X 0,Y 321.27,Z 503.587,A -85,B 0,C 180,E1 -15360.004,E2 -15360.004} C_VEL
LIN {X 0,Y 323.216,Z 505.44,A -85,B 0,C 180,E1 -15360.429,E2 -15360.429} C_VEL
LIN {X 0,Y 325.357,Z 508.702,A -85,B 0,C 180,E1 -15360.966,E2 -15360.966} C_VEL
LIN {X 0,Y 327.418,Z 510.765,A -85,B 0,C 180,E1 -15361.452,E2 -15361.452} C_VEL
LIN {X 0,Y 330.139,Z 514.325,A -85,B 0,C 180,E1 -15362.147,E2 -15362.147} C_VEL
LIN {X 0,Y 332.016,Z 516.342,A -85,B 0,C 180,E1 -15362.614,E2 -15362.614} C_VEL
LIN {X 0,Y 335.082,Z 520.031,A -85,B 0,C 180,E1 -15363.41,E2 -15363.41} C_VEL
LIN {X 0,Y 337.012,Z 522.06,A -85,B 0,C 180,E1 -15363.92,E2 -15363.92} C_VEL
LIN {X 0,Y 340.56,Z 526.033,A -85,B 0,C 180,E1 -15364.882,E2 -15364.882} C_VEL
LIN {X 0,Y 342.481,Z 527.918,A -85,B 0,C 180,E1 -15365.404,E2 -15365.404} C_VEL
LIN {X 0,Y 346.007,Z 531.813,A -85,B 0,C 180,E1 -15366.418,E2 -15366.418} C_VEL
LIN {X 0,Y 348.408,Z 533.999,A -85,B 0,C 180,E1 -15367.109,E2 -15367.109} C_VEL
LIN {X 0,Y 352.305,Z 538.132,A -85,B 0,C 180,E1 -15368.316,E2 -15368.316} C_VEL
LIN {X 0,Y 354.861,Z 540.323,A -85,B 0,C 180,E1 -15369.116,E2 -15369.116} C_VEL
LIN {X 0,Y 358.485,Z 544.113,A -85,B 0,C 180,E1 -15370.34,E2 -15370.34} C_VEL
LIN {X 0,Y 361.922,Z 546.935,A -85,B 0,C 180,E1 -15371.533,E2 -15371.533} C_VEL
LIN {X 0,Y 365.474,Z 550.605,A -85,B 0,C 180,E1 -15372.898,E2 -15372.898} C_VEL
LIN {X 0,Y 369.588,Z 553.734,A -85,B 0,C 180,E1 -15374.561,E2 -15374.561} C_VEL
LIN {X 0,Y 373.034,Z 557.358,A -85,B 0,C 180,E1 -15376.163,E2 -15376.163} C_VEL
LIN {X 0,Y 376.571,Z 559.836,A -85,B 0,C 180,E1 -15377.95,E2 -15377.95} C_VEL
LIN {X 0,Y 378.13,Z 560.774,A -85,B 0,C 180,E1 -15378.812,E2 -15378.812} C_VEL
LIN {X 0,Y 381.153,Z 564.098,A -85,B 0,C 180,E1 -15380.84,E2 -15380.84} C_VEL
LIN {X 0,Y 383.57,Z 565.919,A -85,B 0,C 180,E1 -15382.775,E2 -15382.775} C_VEL
LIN {X 0,Y 385.49,Z 567.027,A -85,B 0,C 180,E1 -15384.77,E2 -15384.77} C_VEL
LIN {X 0,Y 387.015,Z 567.614,A -85,B 0,C 180,E1 -15387.145,E2 -15387.145} C_VEL
LIN {X 0,Y 387.574,Z 567.989,A -85,B 0,C 180,E1 -15388.961,E2 -15388.961} C_VEL
LIN {X 0,Y 387.574,Z 567.992,A -85,B 0,C 180,E1 -15391.039,E2 -15391.039} C_VEL
LIN {X 0,Y 386.892,Z 567.505,A -85,B 0,C 180,E1 -15393.124,E2 -15393.124} C_VEL
LIN {X 0,Y 385.492,Z 567.018,A -85,B 0,C 180,E1 -15395.23,E2 -15395.23} C_VEL
LIN {X 0,Y 383.397,Z 565.813,A -85,B 0,C 180,E1 -15397.372,E2 -15397.372} C_VEL
LIN {X 0,Y 381.027,Z 563.967,A -85,B 0,C 180,E1 -15399.254,E2 -15399.254} C_VEL
LIN {X 0,Y 378.129,Z 560.772,A -85,B 0,C 180,E1 -15401.187,E2 -15401.187} C_VEL
LIN {X 0,Y 374.108,Z 558.217,A -85,B 0,C 180,E1 -15403.308,E2 -15403.308} C_VEL
LIN {X 0,Y 370.627,Z 554.974,A -85,B 0,C 180,E1 -15404.962,E2 -15404.962} C_VEL
LIN {X 0,Y 368.807,Z 553.045,A -85,B 0,C 180,E1 -15405.774,E2 -15405.774} C_VEL
LIN {X 0,Y 364.66,Z 549.865,A -85,B 0,C 180,E1 -15407.425,E2 -15407.425} C_VEL
LIN {X 0,Y 360.721,Z 545.815,A -85,B 0,C 180,E1 -15408.895,E2 -15408.895} C_VEL
LIN {X 0,Y 356.74,Z 542.459,A -85,B 0,C 180,E1 -15410.256,E2 -15410.256} C_VEL
LIN {X 0,Y 353.716,Z 539.263,A -85,B 0,C 180,E1 -15411.251,E2 -15411.251} C_VEL
LIN {X 0,Y 349.801,Z 535.684,A -85,B 0,C 180,E1 -15412.453,E2 -15412.453} C_VEL
LIN {X 0,Y 347.014,Z 532.623,A -85,B 0,C 180,E1 -15413.295,E2 -15413.295} C_VEL
LIN {X 0,Y 343.593,Z 529.345,A -85,B 0,C 180,E1 -15414.27,E2 -15414.27} C_VEL
LIN {X 0,Y 340.908,Z 526.322,A -85,B 0,C 180,E1 -15415.027,E2 -15415.027} C_VEL
LIN {X 0,Y 337.365,Z 522.545,A -85,B 0,C 180,E1 -15415.983,E2 -15415.983} C_VEL
LIN {X 0,Y 335.77,Z 520.657,A -85,B 0,C 180,E1 -15416.412,E2 -15416.412} C_VEL
LIN {X 0,Y 332.546,Z 517.091,A -85,B 0,C 180,E1 -15417.244,E2 -15417.244} C_VEL
LIN {X 0,Y 330.852,Z 514.967,A -85,B 0,C 180,E1 -15417.683,E2 -15417.683} C_VEL
LIN {X 0,Y 328.031,Z 511.721,A -85,B 0,C 180,E1 -15418.389,E2 -15418.389} C_VEL
LIN {X 0,Y 326.788,Z 510.005,A -85,B 0,C 180,E1 -15418.7,E2 -15418.7} C_VEL
LIN {X 0,Y 324.221,Z 507.212,A -85,B 0,C 180,E1 -15419.317,E2 -15419.317} C_VEL
LIN {X 0,Y 322.737,Z 504.869,A -85,B 0,C 180,E1 -15419.679,E2 -15419.679} C_VEL
LIN {X 0,Y 320.641,Z 502.691,A -85,B 0,C 180,E1 -15420.145,E2 -15420.145} C_VEL
LIN {X 0,Y 319.701,Z 500.334,A -85,B 0,C 180,E1 -15420.51,E2 -15420.51} C_VEL
LIN {X 0,Y 319.565,Z 499.829,A -85,B 0,C 180,E1 -15420.942,E2 -15420.942} C_VEL
LIN {X 0,Y 319.554,Z 499.793,A -85,B 0,C 180,E1 -15424.876,E2 -15424.876} C_VEL
LIN {X 0,Y 319.578,Z 499.779,A -85,B 0,C 180,E1 -15428.006,E2 -15428.006} C_VEL
LIN {X 0,Y 319.595,Z 499.766,A -85,B 0,C 180,E1 -15431.612,E2 -15431.612} C_VEL
LIN {X 0,Y 319.639,Z 499.775,A -85,B 0,C 180,E1 -15435.285,E2 -15435.285} C_VEL
LIN {X 0,Y 319.576,Z 499.789,A -85,B 0,C 180,E1 -15438.72,E2 -15438.72} C_VEL
LIN {X 0,Y 319.574,Z 499.799,A -85,B 0,C 180,E1 -15442.343,E2 -15442.343} C_VEL
LIN {X 0,Y 319.553,Z 499.797,A -85,B 0,C 180,E1 -15445.123,E2 -15445.123} C_VEL
LIN {X 0,Y 319.567,Z 499.783,A -85,B 0,C 180,E1 -15449.057,E2 -15449.057} C_VEL
LIN {X 0,Y 319.602,Z 499.8,A -85,B 0,C 180,E1 -15452.498,E2 -15452.498} C_VEL
LIN {X 0,Y 319.597,Z 499.777,A -85,B 0,C 180,E1 -15455.304,E2 -15455.304} C_VEL
LIN {X 0,Y 319.589,Z 499.796,A -85,B 0,C 180,E1 -15458.048,E2 -15458.048} C_VEL
LIN {X 0,Y 319.681,Z 499.776,A -85,B 0,C 180,E1 -15460.963,E2 -15460.963} C_VEL
LIN {X 0,Y 319.723,Z 499.781,A -85,B 0,C 180,E1 -15465.277,E2 -15465.277} C_VEL
LIN {X 0,Y 319.745,Z 499.752,A -85,B 0,C 180,E1 -15469.873,E2 -15469.873} C_VEL
LIN {X 0,Y 319.786,Z 499.749,A -85,B 0,C 180,E1 -15470.752,E2 -15470.752} C_VEL
LIN {X 0,Y 319.51,Z 499.791,A -85,B 0,C 180,E1 -15471.455,E2 -15471.455} C_VEL
LIN {X 0,Y 318.151,Z 499.971,A -85,B 0,C 180,E1 -15472.492,E2 -15472.492} C_VEL
LIN {X 0,Y 313.743,Z 500.522,A -85,B 0,C 180,E1 -15474.898,E2 -15474.898} C_VEL
LIN {X 0,Y 312.755,Z 500.637,A -85,B 0,C 180,E1 -15475.974,E2 -15475.974} C_VEL
LIN {X 0,Y 312.717,Z 500.634,A -85,B 0,C 180,E1 -15476.338,E2 -15476.338} C_VEL
LIN {X 0,Y 312.983,Z 500.594,A -85,B 0,C 180,E1 -15478.714,E2 -15478.714} C_VEL
LIN {X 0,Y 312.983,Z 500.62,A -85,B 0,C 180,E1 -15481.287,E2 -15481.287} C_VEL
LIN {X 0,Y 312.71,Z 500.626,A -85,B 0,C 180,E1 -15485.158,E2 -15485.158} C_VEL
LIN {X 0,Y 312.86,Z 500.628,A -85,B 0,C 180,E1 -15487.747,E2 -15487.747} C_VEL
LIN {X 0,Y 312.662,Z 500.652,A -85,B 0,C 180,E1 -15491.672,E2 -15491.672} C_VEL
LIN {X 0,Y 312.694,Z 500.64,A -85,B 0,C 180,E1 -15494.888,E2 -15494.888} C_VEL
LIN {X 0,Y 312.604,Z 500.657,A -85,B 0,C 180,E1 -15499.226,E2 -15499.226} C_VEL
LIN {X 0,Y 312.521,Z 500.674,A -85,B 0,C 180,E1 -15502.781,E2 -15502.781} C_VEL
LIN {X 0,Y 312.592,Z 500.659,A -85,B 0,C 180,E1 -15505.934,E2 -15505.934} C_VEL
LIN {X 0,Y 312.534,Z 500.678,A -85,B 0,C 180,E1 -15509.652,E2 -15509.652} C_VEL
LIN {X 0,Y 312.516,Z 500.666,A -85,B 0,C 180,E1 -15513.69,E2 -15513.69} C_VEL
LIN {X 0,Y 312.537,Z 500.668,A -85,B 0,C 180,E1 -15517.384,E2 -15517.384} C_VEL
LIN {X 0,Y 312.498,Z 500.683,A -85,B 0,C 180,E1 -15520.709,E2 -15520.709} C_VEL
LIN {X 0,Y 312.463,Z 500.69,A -85,B 0,C 180,E1 -15524.208,E2 -15524.208} C_VEL
LIN {X 0,Y 312.483,Z 500.664,A -85,B 0,C 180,E1 -15527.92,E2 -15527.92} C_VEL
LIN {X 0,Y 312.487,Z 500.715,A -85,B 0,C 180,E1 -15531.632,E2 -15531.632} C_VEL
LIN {X 0,Y 313.086,Z 503.162,A -85,B 0,C 180,E1 -15532.694,E2 -15532.694} C_VEL
LIN {X 0,Y 315.228,Z 512.398,A -85,B 0,C 180,E1 -15536.127,E2 -15536.127} C_VEL
LIN {X 0,Y 316.637,Z 519.198,A -85,B 0,C 180,E1 -15538.498,E2 -15538.498} C_VEL
LIN {X 0,Y 323.356,Z 534.849,A -85,B 0,C 180,E1 -15539.655,E2 -15539.655} C_VEL
LIN {X 0,Y 328.03,Z 556.293,A -85,B 0,C 180,E1 -15540.656,E2 -15540.656} C_VEL
LIN {X 0,Y 330.307,Z 569.031,A -85,B 0,C 180,E1 -15541.186,E2 -15541.186} C_VEL
LIN {X 0,Y 327.862,Z 653.591,A -85,B 0,C 180,E1 -15543.032,E2 -15543.032} C_VEL
LIN {X 0,Y 327.151,Z 664.904,A -85,B 0,C 180,E1 -15543.4,E2 -15543.4} C_VEL
LIN {X 0,Y 326.268,Z 675.446,A -85,B 0,C 180,E1 -15543.882,E2 -15543.882} C_VEL
LIN {X 0,Y 325.038,Z 686.597,A -85,B 0,C 180,E1 -15544.55,E2 -15544.55} C_VEL
LIN {X 0,Y 323.842,Z 696.569,A -85,B 0,C 180,E1 -15545.307,E2 -15545.307} C_VEL
LIN {X 0,Y 322.274,Z 707.239,A -85,B 0,C 180,E1 -15546.295,E2 -15546.295} C_VEL
LIN {X 0,Y 320.968,Z 716.214,A -85,B 0,C 180,E1 -15547.3,E2 -15547.3} C_VEL
LIN {X 0,Y 319.368,Z 725.634,A -85,B 0,C 180,E1 -15548.541,E2 -15548.541} C_VEL
LIN {X 0,Y 317.635,Z 734.652,A -85,B 0,C 180,E1 -15549.944,E2 -15549.944} C_VEL
LIN {X 0,Y 316.389,Z 741.628,A -85,B 0,C 180,E1 -15551.211,E2 -15551.211} C_VEL
LIN {X 0,Y 314.994,Z 749.153,A -85,B 0,C 180,E1 -15552.805,E2 -15552.805} C_VEL
LIN {X 0,Y 313.772,Z 756.247,A -85,B 0,C 180,E1 -15554.589,E2 -15554.589} C_VEL
LIN {X 0,Y 312.812,Z 762.174,A -85,B 0,C 180,E1 -15556.355,E2 -15556.355} C_VEL
LIN {X 0,Y 311.851,Z 767.606,A -85,B 0,C 180,E1 -15558.298,E2 -15558.298} C_VEL
LIN {X 0,Y 311.282,Z 772.053,A -85,B 0,C 180,E1 -15560.251,E2 -15560.251} C_VEL
LIN {X 0,Y 310.959,Z 775.601,A -85,B 0,C 180,E1 -15562.207,E2 -15562.207} C_VEL
LIN {X 0,Y 310.724,Z 778.551,A -85,B 0,C 180,E1 -15564.386,E2 -15564.386} C_VEL
LIN {X 0,Y 310.69,Z 780.23,A -85,B 0,C 180,E1 -15566.109,E2 -15566.109} C_VEL
LIN {X 0,Y 310.656,Z 781.521,A -85,B 0,C 180,E1 -15568.704,E2 -15568.704} C_VEL
LIN {X 0,Y 310.691,Z 781.774,A -85,B 0,C 180,E1 -15570,E2 -15570} C_VEL
LIN {X 0,Y 310.675,Z 781.048,A -85,B 0,C 180,E1 -15572.593,E2 -15572.593} C_VEL
LIN {X 0,Y 310.691,Z 780.23,A -85,B 0,C 180,E1 -15573.891,E2 -15573.891} C_VEL
LIN {X 0,Y 310.813,Z 777.543,A -85,B 0,C 180,E1 -15576.491,E2 -15576.491} C_VEL
LIN {X 0,Y 311.053,Z 774.585,A -85,B 0,C 180,E1 -15578.445,E2 -15578.445} C_VEL
LIN {X 0,Y 311.469,Z 770.755,A -85,B 0,C 180,E1 -15580.399,E2 -15580.399} C_VEL
LIN {X 0,Y 312.167,Z 765.991,A -85,B 0,C 180,E1 -15582.349,E2 -15582.349} C_VEL
LIN {X 0,Y 313.312,Z 759.083,A -85,B 0,C 180,E1 -15584.605,E2 -15584.605} C_VEL
LIN {X 0,Y 314.241,Z 753.168,A -85,B 0,C 180,E1 -15586.233,E2 -15586.233} C_VEL
LIN {X 0,Y 315.509,Z 746.314,A -85,B 0,C 180,E1 -15587.835,E2 -15587.835} C_VEL
LIN {X 0,Y 317.001,Z 738.29,A -85,B 0,C 180,E1 -15589.423,E2 -15589.423} C_VEL
LIN {X 0,Y 318.717,Z 728.81,A -85,B 0,C 180,E1 -15590.997,E2 -15590.997} C_VEL
LIN {X 0,Y 320.38,Z 719.936,A -85,B 0,C 180,E1 -15592.234,E2 -15592.234} C_VEL
LIN {X 0,Y 321.843,Z 710.706,A -85,B 0,C 180,E1 -15593.335,E2 -15593.335} C_VEL
LIN {X 0,Y 323.349,Z 700.076,A -85,B 0,C 180,E1 -15594.391,E2 -15594.391} C_VEL
LIN {X 0,Y 324.657,Z 689.817,A -85,B 0,C 180,E1 -15595.225,E2 -15595.225} C_VEL
LIN {X 0,Y 325.984,Z 678.165,A -85,B 0,C 180,E1 -15595.971,E2 -15595.971} C_VEL
LIN {X 0,Y 326.965,Z 667.641,A -85,B 0,C 180,E1 -15596.488,E2 -15596.488} C_VEL
LIN {X 0,Y 327.72,Z 656.226,A -85,B 0,C 180,E1 -15596.894,E2 -15596.894} C_VEL
LIN {X 0,Y 328.718,Z 626.115,A -85,B 0,C 180,E1 -15597.581,E2 -15597.581} C_VEL
LIN {X 0,Y 330.211,Z 567.807,A -85,B 0,C 180,E1 -15598.853,E2 -15598.853} C_VEL
LIN {X 0,Y 325.326,Z 543.048,A -85,B 0,C 180,E1 -15599.939,E2 -15599.939} C_VEL
LIN {X 0,Y 323.074,Z 534.137,A -85,B 0,C 180,E1 -15600.392,E2 -15600.392} C_VEL
LIN {X 0,Y 316.645,Z 519.181,A -85,B 0,C 180,E1 -15601.503,E2 -15601.503} C_VEL
LIN {X 0,Y 314.666,Z 509.791,A -85,B 0,C 180,E1 -15604.832,E2 -15604.832} C_VEL
LIN {X 0,Y 312.526,Z 500.878,A -85,B 0,C 180,E1 -15608.23,E2 -15608.23} C_VEL
LIN {X 0,Y 312.503,Z 500.676,A -85,B 0,C 180,E1 -15610.124,E2 -15610.124} C_VEL
LIN {X 0,Y 312.457,Z 500.661,A -85,B 0,C 180,E1 -15613.964,E2 -15613.964} C_VEL
LIN {X 0,Y 312.525,Z 500.671,A -85,B 0,C 180,E1 -15617.909,E2 -15617.909} C_VEL
LIN {X 0,Y 312.54,Z 500.665,A -85,B 0,C 180,E1 -15621.908,E2 -15621.908} C_VEL
LIN {X 0,Y 312.503,Z 500.673,A -85,B 0,C 180,E1 -15625.789,E2 -15625.789} C_VEL
LIN {X 0,Y 312.516,Z 500.677,A -85,B 0,C 180,E1 -15628.853,E2 -15628.853} C_VEL
LIN {X 0,Y 312.565,Z 500.659,A -85,B 0,C 180,E1 -15631.823,E2 -15631.823} C_VEL
LIN {X 0,Y 312.58,Z 500.667,A -85,B 0,C 180,E1 -15634.71,E2 -15634.71} C_VEL
LIN {X 0,Y 312.531,Z 500.656,A -85,B 0,C 180,E1 -15638.912,E2 -15638.912} C_VEL
LIN {X 0,Y 312.633,Z 500.661,A -85,B 0,C 180,E1 -15641.655,E2 -15641.655} C_VEL
LIN {X 0,Y 312.688,Z 500.633,A -85,B 0,C 180,E1 -15645.685,E2 -15645.685} C_VEL
LIN {X 0,Y 312.695,Z 500.659,A -85,B 0,C 180,E1 -15649.641,E2 -15649.641} C_VEL
LIN {X 0,Y 312.86,Z 500.628,A -85,B 0,C 180,E1 -15652.253,E2 -15652.253} C_VEL
LIN {X 0,Y 312.709,Z 500.626,A -85,B 0,C 180,E1 -15654.842,E2 -15654.842} C_VEL
LIN {X 0,Y 312.983,Z 500.62,A -85,B 0,C 180,E1 -15658.713,E2 -15658.713} C_VEL
LIN {X 0,Y 312.983,Z 500.594,A -85,B 0,C 180,E1 -15661.286,E2 -15661.286} C_VEL
LIN {X 0,Y 312.709,Z 500.652,A -85,B 0,C 180,E1 -15665.157,E2 -15665.157} C_VEL
LIN {X 0,Y 312.846,Z 500.628,A -85,B 0,C 180,E1 -15667.746,E2 -15667.746} C_VEL
LIN {X 0,Y 312.661,Z 500.648,A -85,B 0,C 180,E1 -15671.671,E2 -15671.671} C_VEL
LIN {X 0,Y 312.693,Z 500.658,A -85,B 0,C 180,E1 -15674.887,E2 -15674.887} C_VEL
LIN {X 0,Y 312.623,Z 500.657,A -85,B 0,C 180,E1 -15679.236,E2 -15679.236} C_VEL
LIN {X 0,Y 312.538,Z 500.667,A -85,B 0,C 180,E1 -15682.789,E2 -15682.789} C_VEL
LIN {X 0,Y 312.595,Z 500.66,A -85,B 0,C 180,E1 -15685.935,E2 -15685.935} C_VEL
LIN {X 0,Y 312.539,Z 500.661,A -85,B 0,C 180,E1 -15689.65,E2 -15689.65} C_VEL
LIN {X 0,Y 312.513,Z 500.683,A -85,B 0,C 180,E1 -15693.689,E2 -15693.689} C_VEL
LIN {X 0,Y 312.533,Z 500.673,A -85,B 0,C 180,E1 -15697.383,E2 -15697.383} C_VEL
LIN {X 0,Y 312.521,Z 500.666,A -85,B 0,C 180,E1 -15700.703,E2 -15700.703} C_VEL
LIN {X 0,Y 312.589,Z 500.665,A -85,B 0,C 180,E1 -15704.184,E2 -15704.184} C_VEL
LIN {X 0,Y 312.55,Z 500.635,A -85,B 0,C 180,E1 -15707.904,E2 -15707.904} C_VEL
LIN {X 0,Y 312.539,Z 500.656,A -85,B 0,C 180,E1 -15711.908,E2 -15711.908} C_VEL
LIN {X 0,Y 312.501,Z 500.685,A -85,B 0,C 180,E1 -15715.79,E2 -15715.79} C_VEL
LIN {X 0,Y 312.538,Z 500.903,A -85,B 0,C 180,E1 -15718.147,E2 -15718.147} C_VEL
LIN {X 0,Y 312.823,Z 502.066,A -85,B 0,C 180,E1 -15718.428,E2 -15718.428} C_VEL
LIN {X 0,Y 314.508,Z 504.824,A -85,B 0,C 180,E1 -15718.823,E2 -15718.823} C_VEL
LIN {X 0,Y 315.848,Z 506.165,A -85,B 0,C 180,E1 -15719.092,E2 -15719.092} C_VEL
LIN {X 0,Y 318.055,Z 509.442,A -85,B 0,C 180,E1 -15719.576,E2 -15719.576} C_VEL
LIN {X 0,Y 319.905,Z 511.464,A -85,B 0,C 180,E1 -15719.997,E2 -15719.997} C_VEL
LIN {X 0,Y 322.612,Z 514.977,A -85,B 0,C 180,E1 -15720.619,E2 -15720.619} C_VEL
LIN {X 0,Y 324.487,Z 517.038,A -85,B 0,C 180,E1 -15721.064,E2 -15721.064} C_VEL
LIN {X 0,Y 328.024,Z 521.113,A -85,B 0,C 180,E1 -15721.927,E2 -15721.927} C_VEL
LIN {X 0,Y 332.318,Z 526.156,A -85,B 0,C 180,E1 -15723.017,E2 -15723.017} C_VEL
LIN {X 0,Y 334.349,Z 528.294,A -85,B 0,C 180,E1 -15723.532,E2 -15723.532} C_VEL
LIN {X 0,Y 338.237,Z 532.47,A -85,B 0,C 180,E1 -15724.562,E2 -15724.562} C_VEL
LIN {X 0,Y 343.842,Z 538.321,A -85,B 0,C 180,E1 -15726.114,E2 -15726.114} C_VEL
LIN {X 0,Y 346.534,Z 540.919,A -85,B 0,C 180,E1 -15726.891,E2 -15726.891} C_VEL
LIN {X 0,Y 350.538,Z 544.888,A -85,B 0,C 180,E1 -15728.091,E2 -15728.091} C_VEL
LIN {X 0,Y 352.963,Z 547.047,A -85,B 0,C 180,E1 -15728.847,E2 -15728.847} C_VEL
LIN {X 0,Y 356.682,Z 550.775,A -85,B 0,C 180,E1 -15730.074,E2 -15730.074} C_VEL
LIN {X 0,Y 360.2,Z 553.685,A -85,B 0,C 180,E1 -15731.283,E2 -15731.283} C_VEL
LIN {X 0,Y 363.85,Z 557.323,A -85,B 0,C 180,E1 -15732.643,E2 -15732.643} C_VEL
LIN {X 0,Y 368.143,Z 560.643,A -85,B 0,C 180,E1 -15734.354,E2 -15734.354} C_VEL
LIN {X 0,Y 371.678,Z 564.218,A -85,B 0,C 180,E1 -15735.972,E2 -15735.972} C_VEL
LIN {X 0,Y 374.992,Z 566.52,A -85,B 0,C 180,E1 -15737.6,E2 -15737.6} C_VEL
LIN {X 0,Y 377.021,Z 567.823,A -85,B 0,C 180,E1 -15738.704,E2 -15738.704} C_VEL
LIN {X 0,Y 380.091,Z 571.077,A -85,B 0,C 180,E1 -15740.721,E2 -15740.721} C_VEL
LIN {X 0,Y 382.604,Z 572.929,A -85,B 0,C 180,E1 -15742.705,E2 -15742.705} C_VEL
LIN {X 0,Y 384.608,Z 574.047,A -85,B 0,C 180,E1 -15744.758,E2 -15744.758} C_VEL
LIN {X 0,Y 386.02,Z 574.557,A -85,B 0,C 180,E1 -15746.869,E2 -15746.869} C_VEL
LIN {X 0,Y 386.708,Z 575.035,A -85,B 0,C 180,E1 -15748.959,E2 -15748.959} C_VEL
LIN {X 0,Y 386.708,Z 575.038,A -85,B 0,C 180,E1 -15751.041,E2 -15751.041} C_VEL
LIN {X 0,Y 386.02,Z 574.557,A -85,B 0,C 180,E1 -15753.131,E2 -15753.131} C_VEL
LIN {X 0,Y 384.606,Z 574.067,A -85,B 0,C 180,E1 -15755.242,E2 -15755.242} C_VEL
LIN {X 0,Y 382.491,Z 572.861,A -85,B 0,C 180,E1 -15757.39,E2 -15757.39} C_VEL
LIN {X 0,Y 379.878,Z 570.883,A -85,B 0,C 180,E1 -15759.423,E2 -15759.423} C_VEL
LIN {X 0,Y 376.886,Z 567.677,A -85,B 0,C 180,E1 -15761.375,E2 -15761.375} C_VEL
LIN {X 0,Y 372.956,Z 565.206,A -85,B 0,C 180,E1 -15763.421,E2 -15763.421} C_VEL
LIN {X 0,Y 369.265,Z 561.895,A -85,B 0,C 180,E1 -15765.14,E2 -15765.14} C_VEL
LIN {X 0,Y 367,Z 559.598,A -85,B 0,C 180,E1 -15766.121,E2 -15766.121} C_VEL
LIN {X 0,Y 362.786,Z 556.401,A -85,B 0,C 180,E1 -15767.754,E2 -15767.754} C_VEL
LIN {X 0,Y 358.8,Z 552.362,A -85,B 0,C 180,E1 -15769.22,E2 -15769.22} C_VEL
LIN {X 0,Y 354.615,Z 548.874,A -85,B 0,C 180,E1 -15770.606,E2 -15770.606} C_VEL
LIN {X 0,Y 351.425,Z 545.587,A -85,B 0,C 180,E1 -15771.634,E2 -15771.634} C_VEL
LIN {X 0,Y 347.345,Z 541.864,A -85,B 0,C 180,E1 -15772.869,E2 -15772.869} C_VEL
LIN {X 0,Y 344.382,Z 538.762,A -85,B 0,C 180,E1 -15773.737,E2 -15773.737} C_VEL
LIN {X 0,Y 340.2,Z 534.552,A -85,B 0,C 180,E1 -15774.902,E2 -15774.902} C_VEL
LIN {X 0,Y 337.473,Z 531.744,A -85,B 0,C 180,E1 -15775.642,E2 -15775.642} C_VEL
LIN {X 0,Y 333.733,Z 527.452,A -85,B 0,C 180,E1 -15776.633,E2 -15776.633} C_VEL
LIN {X 0,Y 329.667,Z 523.202,A -85,B 0,C 180,E1 -15777.656,E2 -15777.656} C_VEL
LIN {X 0,Y 327.9,Z 520.992,A -85,B 0,C 180,E1 -15778.103,E2 -15778.103} C_VEL
LIN {X 0,Y 324.583,Z 517.15,A -85,B 0,C 180,E1 -15778.913,E2 -15778.913} C_VEL
LIN {X 0,Y 323.269,Z 515.593,A -85,B 0,C 180,E1 -15779.231,E2 -15779.231} C_VEL
LIN {X 0,Y 320.24,Z 512.043,A -85,B 0,C 180,E1 -15779.923,E2 -15779.923} C_VEL
LIN {X 0,Y 318.87,Z 510.264,A -85,B 0,C 180,E1 -15780.243,E2 -15780.243} C_VEL
LIN {X 0,Y 316.426,Z 507.223,A -85,B 0,C 180,E1 -15780.779,E2 -15780.779} C_VEL
LIN {X 0,Y 315.125,Z 505.353,A -85,B 0,C 180,E1 -15781.056,E2 -15781.056} C_VEL
LIN {X 0,Y 313.143,Z 502.903,A -85,B 0,C 180,E1 -15781.479,E2 -15781.479} C_VEL
LIN {X 0,Y 312.574,Z 501.235,A -85,B 0,C 180,E1 -15781.721,E2 -15781.721} C_VEL
LIN {X 0,Y 312.481,Z 500.718,A -85,B 0,C 180,E1 -15782.105,E2 -15782.105} C_VEL
LIN {X 0,Y 312.53,Z 500.65,A -85,B 0,C 180,E1 -15785.949,E2 -15785.949} C_VEL
LIN {X 0,Y 312.528,Z 500.676,A -85,B 0,C 180,E1 -15789.023,E2 -15789.023} C_VEL
LIN {X 0,Y 312.554,Z 500.631,A -85,B 0,C 180,E1 -15792.42,E2 -15792.42} C_VEL
LIN {X 0,Y 312.586,Z 500.667,A -85,B 0,C 180,E1 -15796.009,E2 -15796.009} C_VEL
LIN {X 0,Y 312.524,Z 500.669,A -85,B 0,C 180,E1 -15799.869,E2 -15799.869} C_VEL
LIN {X 0,Y 312.533,Z 500.673,A -85,B 0,C 180,E1 -15802.617,E2 -15802.617} C_VEL
LIN {X 0,Y 312.513,Z 500.683,A -85,B 0,C 180,E1 -15806.311,E2 -15806.311} C_VEL
LIN {X 0,Y 312.539,Z 500.661,A -85,B 0,C 180,E1 -15810.35,E2 -15810.35} C_VEL
LIN {X 0,Y 312.595,Z 500.66,A -85,B 0,C 180,E1 -15814.065,E2 -15814.065} C_VEL
LIN {X 0,Y 312.58,Z 500.666,A -85,B 0,C 180,E1 -15817.529,E2 -15817.529} C_VEL
LIN {X 0,Y 312.63,Z 500.646,A -85,B 0,C 180,E1 -15821.657,E2 -15821.657} C_VEL
LIN {X 0,Y 312.686,Z 500.658,A -85,B 0,C 180,E1 -15825.687,E2 -15825.687} C_VEL
LIN {X 0,Y 312.691,Z 500.631,A -85,B 0,C 180,E1 -15829.642,E2 -15829.642} C_VEL
LIN {X 0,Y 312.847,Z 500.628,A -85,B 0,C 180,E1 -15832.254,E2 -15832.254} C_VEL
LIN {X 0,Y 312.712,Z 500.651,A -85,B 0,C 180,E1 -15834.843,E2 -15834.843} C_VEL
LIN {X 0,Y 312.717,Z 500.634,A -85,B 0,C 180,E1 -15836.338,E2 -15836.338} C_VEL
LIN {X 0,Y 312.186,Z 500.692,A -85,B 0,C 180,E1 -15837.416,E2 -15837.416} C_VEL
LIN {X 0,Y 309.45,Z 501.039,A -85,B 0,C 180,E1 -15839.174,E2 -15839.174} C_VEL
LIN {X 0,Y 307.045,Z 501.355,A -85,B 0,C 180,E1 -15840.599,E2 -15840.599} C_VEL
LIN {X 0,Y 305.986,Z 501.491,A -85,B 0,C 180,E1 -15841.701,E2 -15841.701} C_VEL
LIN {X 0,Y 305.89,Z 501.5,A -85,B 0,C 180,E1 -15842.075,E2 -15842.075} C_VEL
LIN {X 0,Y 305.841,Z 501.484,A -85,B 0,C 180,E1 -15846.598,E2 -15846.598} C_VEL
LIN {X 0,Y 305.73,Z 501.526,A -85,B 0,C 180,E1 -15849.261,E2 -15849.261} C_VEL
LIN {X 0,Y 305.581,Z 501.514,A -85,B 0,C 180,E1 -15853.297,E2 -15853.297} C_VEL
LIN {X 0,Y 305.588,Z 501.539,A -85,B 0,C 180,E1 -15856.021,E2 -15856.021} C_VEL
LIN {X 0,Y 305.555,Z 501.531,A -85,B 0,C 180,E1 -15859.437,E2 -15859.437} C_VEL
LIN {X 0,Y 305.481,Z 501.554,A -85,B 0,C 180,E1 -15863.04,E2 -15863.04} C_VEL
LIN {X 0,Y 305.521,Z 501.535,A -85,B 0,C 180,E1 -15866.219,E2 -15866.219} C_VEL
LIN {X 0,Y 305.484,Z 501.551,A -85,B 0,C 180,E1 -15869.048,E2 -15869.048} C_VEL
LIN {X 0,Y 305.438,Z 501.552,A -85,B 0,C 180,E1 -15871.953,E2 -15871.953} C_VEL
LIN {X 0,Y 305.459,Z 501.56,A -85,B 0,C 180,E1 -15875.114,E2 -15875.114} C_VEL
LIN {X 0,Y 305.479,Z 501.547,A -85,B 0,C 180,E1 -15878.537,E2 -15878.537} C_VEL
LIN {X 0,Y 305.484,Z 501.551,A -85,B 0,C 180,E1 -15882.593,E2 -15882.593} C_VEL
LIN {X 0,Y 305.453,Z 501.533,A -85,B 0,C 180,E1 -15887.415,E2 -15887.415} C_VEL
LIN {X 0,Y 305.468,Z 501.66,A -85,B 0,C 180,E1 -15891.062,E2 -15891.062} C_VEL
LIN {X 0,Y 307.435,Z 509.878,A -85,B 0,C 180,E1 -15894.344,E2 -15894.344} C_VEL
LIN {X 0,Y 309.346,Z 518.783,A -85,B 0,C 180,E1 -15897.639,E2 -15897.639} C_VEL
LIN {X 0,Y 311.212,Z 523.096,A -85,B 0,C 180,E1 -15898.036,E2 -15898.036} C_VEL
LIN {X 0,Y 317.666,Z 538.096,A -85,B 0,C 180,E1 -15899.141,E2 -15899.141} C_VEL
LIN {X 0,Y 322.13,Z 559.075,A -85,B 0,C 180,E1 -15900.139,E2 -15900.139} C_VEL
LIN {X 0,Y 324.065,Z 570.173,A -85,B 0,C 180,E1 -15900.61,E2 -15900.61} C_VEL
LIN {X 0,Y 321.498,Z 654.705,A -85,B 0,C 180,E1 -15902.498,E2 -15902.498} C_VEL
LIN {X 0,Y 320.758,Z 665.618,A -85,B 0,C 180,E1 -15902.87,E2 -15902.87} C_VEL
LIN {X 0,Y 319.757,Z 676.607,A -85,B 0,C 180,E1 -15903.396,E2 -15903.396} C_VEL
LIN {X 0,Y 318.638,Z 686.399,A -85,B 0,C 180,E1 -15904.001,E2 -15904.001} C_VEL
LIN {X 0,Y 317.39,Z 696.37,A -85,B 0,C 180,E1 -15904.771,E2 -15904.771} C_VEL
LIN {X 0,Y 315.825,Z 706.685,A -85,B 0,C 180,E1 -15905.738,E2 -15905.738} C_VEL
LIN {X 0,Y 314.407,Z 716.016,A -85,B 0,C 180,E1 -15906.799,E2 -15906.799} C_VEL
LIN {X 0,Y 312.746,Z 725.435,A -85,B 0,C 180,E1 -15908.063,E2 -15908.063} C_VEL
LIN {X 0,Y 310.924,Z 734.452,A -85,B 0,C 180,E1 -15909.491,E2 -15909.491} C_VEL
LIN {X 0,Y 309.64,Z 741.429,A -85,B 0,C 180,E1 -15910.786,E2 -15910.786} C_VEL
LIN {X 0,Y 308.153,Z 748.953,A -85,B 0,C 180,E1 -15912.411,E2 -15912.411} C_VEL
LIN {X 0,Y 306.876,Z 755.695,A -85,B 0,C 180,E1 -15914.129,E2 -15914.129} C_VEL
LIN {X 0,Y 305.855,Z 761.974,A -85,B 0,C 180,E1 -15916.039,E2 -15916.039} C_VEL
LIN {X 0,Y 304.861,Z 767.406,A -85,B 0,C 180,E1 -15918.026,E2 -15918.026} C_VEL
LIN {X 0,Y 304.26,Z 771.854,A -85,B 0,C 180,E1 -15920.024,E2 -15920.024} C_VEL
LIN {X 0,Y 303.881,Z 775.402,A -85,B 0,C 180,E1 -15922.024,E2 -15922.024} C_VEL
LIN {X 0,Y 303.724,Z 777.344,A -85,B 0,C 180,E1 -15923.356,E2 -15923.356} C_VEL
LIN {X 0,Y 303.586,Z 780.031,A -85,B 0,C 180,E1 -15926.018,E2 -15926.018} C_VEL
LIN {X 0,Y 303.573,Z 781.323,A -85,B 0,C 180,E1 -15928.673,E2 -15928.673} C_VEL
LIN {X 0,Y 303.604,Z 781.576,A -85,B 0,C 180,E1 -15930,E2 -15930} C_VEL
LIN {X 0,Y 303.6,Z 780.85,A -85,B 0,C 180,E1 -15932.654,E2 -15932.654} C_VEL
LIN {X 0,Y 303.587,Z 780.031,A -85,B 0,C 180,E1 -15933.982,E2 -15933.982} C_VEL
LIN {X 0,Y 303.725,Z 777.344,A -85,B 0,C 180,E1 -15936.644,E2 -15936.644} C_VEL
LIN {X 0,Y 303.987,Z 774.385,A -85,B 0,C 180,E1 -15938.643,E2 -15938.643} C_VEL
LIN {X 0,Y 304.437,Z 770.556,A -85,B 0,C 180,E1 -15940.642,E2 -15940.642} C_VEL
LIN {X 0,Y 305.198,Z 765.792,A -85,B 0,C 180,E1 -15942.636,E2 -15942.636} C_VEL
LIN {X 0,Y 306.398,Z 758.936,A -85,B 0,C 180,E1 -15944.927,E2 -15944.927} C_VEL
LIN {X 0,Y 307.396,Z 752.967,A -85,B 0,C 180,E1 -15946.606,E2 -15946.606} C_VEL
LIN {X 0,Y 309.015,Z 744.553,A -85,B 0,C 180,E1 -15948.566,E2 -15948.566} C_VEL
LIN {X 0,Y 310.581,Z 736.271,A -85,B 0,C 180,E1 -15950.187,E2 -15950.187} C_VEL
LIN {X 0,Y 312.297,Z 727.552,A -85,B 0,C 180,E1 -15951.623,E2 -15951.623} C_VEL
LIN {X 0,Y 314.038,Z 718.498,A -85,B 0,C 180,E1 -15952.882,E2 -15952.882} C_VEL
LIN {X 0,Y 315.335,Z 710.249,A -85,B 0,C 180,E1 -15953.877,E2 -15953.877} C_VEL
LIN {X 0,Y 316.871,Z 699.877,A -85,B 0,C 180,E1 -15954.923,E2 -15954.923} C_VEL
LIN {X 0,Y 318.228,Z 689.619,A -85,B 0,C 180,E1 -15955.772,E2 -15955.772} C_VEL
LIN {X 0,Y 319.616,Z 677.967,A -85,B 0,C 180,E1 -15956.528,E2 -15956.528} C_VEL
LIN {X 0,Y 320.697,Z 666.531,A -85,B 0,C 180,E1 -15957.091,E2 -15957.091} C_VEL
LIN {X 0,Y 321.408,Z 656.029,A -85,B 0,C 180,E1 -15957.467,E2 -15957.467} C_VEL
LIN {X 0,Y 322.443,Z 625.917,A -85,B 0,C 180,E1 -15958.165,E2 -15958.165} C_VEL
LIN {X 0,Y 324.002,Z 568.951,A -85,B 0,C 180,E1 -15959.426,E2 -15959.426} C_VEL
LIN {X 0,Y 318.992,Z 543.562,A -85,B 0,C 180,E1 -15960.578,E2 -15960.578} C_VEL
LIN {X 0,Y 317.202,Z 536.821,A -85,B 0,C 180,E1 -15960.942,E2 -15960.942} C_VEL
LIN {X 0,Y 309.401,Z 518.946,A -85,B 0,C 180,E1 -15962.328,E2 -15962.328} C_VEL
LIN {X 0,Y 307.964,Z 512.154,A -85,B 0,C 180,E1 -15964.786,E2 -15964.786} C_VEL
LIN {X 0,Y 306.075,Z 504.143,A -85,B 0,C 180,E1 -15967.894,E2 -15967.894} C_VEL
LIN {X 0,Y 305.447,Z 501.563,A -85,B 0,C 180,E1 -15969.02,E2 -15969.02} C_VEL
LIN {X 0,Y 305.453,Z 501.532,A -85,B 0,C 180,E1 -15972.585,E2 -15972.585} C_VEL
LIN {X 0,Y 305.484,Z 501.549,A -85,B 0,C 180,E1 -15977.407,E2 -15977.407} C_VEL
LIN {X 0,Y 305.505,Z 501.542,A -85,B 0,C 180,E1 -15981.601,E2 -15981.601} C_VEL
LIN {X 0,Y 305.459,Z 501.56,A -85,B 0,C 180,E1 -15984.886,E2 -15984.886} C_VEL
LIN {X 0,Y 305.445,Z 501.555,A -85,B 0,C 180,E1 -15988.355,E2 -15988.355} C_VEL
LIN {X 0,Y 305.509,Z 501.545,A -85,B 0,C 180,E1 -15991.112,E2 -15991.112} C_VEL
LIN {X 0,Y 305.56,Z 501.535,A -85,B 0,C 180,E1 -15994.086,E2 -15994.086} C_VEL
LIN {X 0,Y 305.476,Z 501.538,A -85,B 0,C 180,E1 -15998.4,E2 -15998.4} C_VEL
LIN {X 0,Y 305.574,Z 501.535,A -85,B 0,C 180,E1 -16001.216,E2 -16001.216} C_VEL
LIN {X 0,Y 305.643,Z 501.514,A -85,B 0,C 180,E1 -16005.348,E2 -16005.348} C_VEL
LIN {X 0,Y 305.631,Z 501.536,A -85,B 0,C 180,E1 -16009.399,E2 -16009.399} C_VEL
LIN {X 0,Y 305.802,Z 501.508,A -85,B 0,C 180,E1 -16012.073,E2 -16012.073} C_VEL
LIN {X 0,Y 305.681,Z 501.5,A -85,B 0,C 180,E1 -16014.723,E2 -16014.723} C_VEL
LIN {X 0,Y 305.95,Z 501.496,A -85,B 0,C 180,E1 -16018.683,E2 -16018.683} C_VEL
LIN {X 0,Y 305.95,Z 501.469,A -85,B 0,C 180,E1 -16021.316,E2 -16021.316} C_VEL
LIN {X 0,Y 305.68,Z 501.528,A -85,B 0,C 180,E1 -16025.276,E2 -16025.276} C_VEL
LIN {X 0,Y 305.789,Z 501.505,A -85,B 0,C 180,E1 -16027.926,E2 -16027.926} C_VEL
LIN {X 0,Y 305.596,Z 501.531,A -85,B 0,C 180,E1 -16031.945,E2 -16031.945} C_VEL
LIN {X 0,Y 305.63,Z 501.534,A -85,B 0,C 180,E1 -16035.034,E2 -16035.034} C_VEL
LIN {X 0,Y 305.569,Z 501.537,A -85,B 0,C 180,E1 -16039.444,E2 -16039.444} C_VEL
LIN {X 0,Y 305.483,Z 501.541,A -85,B 0,C 180,E1 -16043.041,E2 -16043.041} C_VEL
LIN {X 0,Y 305.54,Z 501.543,A -85,B 0,C 180,E1 -16046.227,E2 -16046.227} C_VEL
LIN {X 0,Y 305.489,Z 501.547,A -85,B 0,C 180,E1 -16049.05,E2 -16049.05} C_VEL
LIN {X 0,Y 305.44,Z 501.552,A -85,B 0,C 180,E1 -16051.952,E2 -16051.952} C_VEL
LIN {X 0,Y 305.455,Z 501.549,A -85,B 0,C 180,E1 -16055.113,E2 -16055.113} C_VEL
LIN {X 0,Y 305.485,Z 501.558,A -85,B 0,C 180,E1 -16058.539,E2 -16058.539} C_VEL
LIN {X 0,Y 305.516,Z 501.555,A -85,B 0,C 180,E1 -16062.6,E2 -16062.6} C_VEL
LIN {X 0,Y 305.527,Z 501.504,A -85,B 0,C 180,E1 -16066.364,E2 -16066.364} C_VEL
LIN {X 0,Y 305.494,Z 501.555,A -85,B 0,C 180,E1 -16069.899,E2 -16069.899} C_VEL
LIN {X 0,Y 305.494,Z 501.523,A -85,B 0,C 180,E1 -16073.627,E2 -16073.627} C_VEL
LIN {X 0,Y 305.494,Z 501.712,A -85,B 0,C 180,E1 -16077.04,E2 -16077.04} C_VEL
LIN {X 0,Y 305.69,Z 502.656,A -85,B 0,C 180,E1 -16077.315,E2 -16077.315} C_VEL
LIN {X 0,Y 307.222,Z 505.434,A -85,B 0,C 180,E1 -16077.667,E2 -16077.667} C_VEL
LIN {X 0,Y 308.483,Z 507.081,A -85,B 0,C 180,E1 -16077.909,E2 -16077.909} C_VEL
LIN {X 0,Y 310.985,Z 510.531,A -85,B 0,C 180,E1 -16078.396,E2 -16078.396} C_VEL
LIN {X 0,Y 312.614,Z 512.654,A -85,B 0,C 180,E1 -16078.74,E2 -16078.74} C_VEL
LIN {X 0,Y 315.734,Z 516.262,A -85,B 0,C 180,E1 -16079.382,E2 -16079.382} C_VEL
LIN {X 0,Y 319.286,Z 520.751,A -85,B 0,C 180,E1 -16080.178,E2 -16080.178} C_VEL
LIN {X 0,Y 321.68,Z 523.44,A -85,B 0,C 180,E1 -16080.713,E2 -16080.713} C_VEL
LIN {X 0,Y 327.305,Z 529.912,A -85,B 0,C 180,E1 -16082.072,E2 -16082.072} C_VEL
LIN {X 0,Y 332.196,Z 535.204,A -85,B 0,C 180,E1 -16083.298,E2 -16083.298} C_VEL
LIN {X 0,Y 337.861,Z 541.082,A -85,B 0,C 180,E1 -16084.781,E2 -16084.781} C_VEL
LIN {X 0,Y 342.516,Z 545.553,A -85,B 0,C 180,E1 -16086.054,E2 -16086.054} C_VEL
LIN {X 0,Y 347.982,Z 551.049,A -85,B 0,C 180,E1 -16087.652,E2 -16087.652} C_VEL
LIN {X 0,Y 350.753,Z 553.449,A -85,B 0,C 180,E1 -16088.49,E2 -16088.49} C_VEL
LIN {X 0,Y 354.789,Z 557.381,A -85,B 0,C 180,E1 -16089.787,E2 -16089.787} C_VEL
LIN {X 0,Y 358.32,Z 560.279,A -85,B 0,C 180,E1 -16090.973,E2 -16090.973} C_VEL
LIN {X 0,Y 362.377,Z 564.184,A -85,B 0,C 180,E1 -16092.462,E2 -16092.462} C_VEL
LIN {X 0,Y 366.451,Z 567.275,A -85,B 0,C 180,E1 -16094.056,E2 -16094.056} C_VEL
LIN {X 0,Y 370.182,Z 570.954,A -85,B 0,C 180,E1 -16095.712,E2 -16095.712} C_VEL
LIN {X 0,Y 373.786,Z 573.44,A -85,B 0,C 180,E1 -16097.445,E2 -16097.445} C_VEL
LIN {X 0,Y 375.776,Z 574.737,A -85,B 0,C 180,E1 -16098.515,E2 -16098.515} C_VEL
LIN {X 0,Y 379.015,Z 578.049,A -85,B 0,C 180,E1 -16100.602,E2 -16100.602} C_VEL
LIN {X 0,Y 381.582,Z 579.92,A -85,B 0,C 180,E1 -16102.593,E2 -16102.593} C_VEL
LIN {X 0,Y 383.723,Z 581.094,A -85,B 0,C 180,E1 -16104.746,E2 -16104.746} C_VEL
LIN {X 0,Y 385.148,Z 581.607,A -85,B 0,C 180,E1 -16106.862,E2 -16106.862} C_VEL
LIN {X 0,Y 385.842,Z 582.081,A -85,B 0,C 180,E1 -16108.956,E2 -16108.956} C_VEL
LIN {X 0,Y 385.842,Z 582.084,A -85,B 0,C 180,E1 -16111.044,E2 -16111.044} C_VEL
LIN {X 0,Y 385.148,Z 581.606,A -85,B 0,C 180,E1 -16113.138,E2 -16113.138} C_VEL
LIN {X 0,Y 383.721,Z 581.116,A -85,B 0,C 180,E1 -16115.254,E2 -16115.254} C_VEL
LIN {X 0,Y 381.585,Z 579.907,A -85,B 0,C 180,E1 -16117.407,E2 -16117.407} C_VEL
LIN {X 0,Y 378.944,Z 577.982,A -85,B 0,C 180,E1 -16119.446,E2 -16119.446} C_VEL
LIN {X 0,Y 375.777,Z 574.721,A -85,B 0,C 180,E1 -16121.485,E2 -16121.485} C_VEL
LIN {X 0,Y 371.488,Z 571.959,A -85,B 0,C 180,E1 -16123.685,E2 -16123.685} C_VEL
LIN {X 0,Y 367.787,Z 568.685,A -85,B 0,C 180,E1 -16125.372,E2 -16125.372} C_VEL
LIN {X 0,Y 365.492,Z 566.408,A -85,B 0,C 180,E1 -16126.346,E2 -16126.346} C_VEL
LIN {X 0,Y 361.117,Z 563.115,A -85,B 0,C 180,E1 -16128.006,E2 -16128.006} C_VEL
LIN {X 0,Y 356.649,Z 558.803,A -85,B 0,C 180,E1 -16129.598,E2 -16129.598} C_VEL
LIN {X 0,Y 352.382,Z 555.172,A -85,B 0,C 180,E1 -16130.995,E2 -16130.995} C_VEL
LIN {X 0,Y 349.138,Z 551.94,A -85,B 0,C 180,E1 -16132.009,E2 -16132.009} C_VEL
LIN {X 0,Y 344.799,Z 547.981,A -85,B 0,C 180,E1 -16133.286,E2 -16133.286} C_VEL
LIN {X 0,Y 341.656,Z 544.822,A -85,B 0,C 180,E1 -16134.182,E2 -16134.182} C_VEL
LIN {X 0,Y 337.48,Z 540.611,A -85,B 0,C 180,E1 -16135.326,E2 -16135.326} C_VEL
LIN {X 0,Y 331.659,Z 534.563,A -85,B 0,C 180,E1 -16136.84,E2 -16136.84} C_VEL
LIN {X 0,Y 326.067,Z 528.356,A -85,B 0,C 180,E1 -16138.241,E2 -16138.241} C_VEL
LIN {X 0,Y 321.319,Z 522.874,A -85,B 0,C 180,E1 -16139.378,E2 -16139.378} C_VEL
LIN {X 0,Y 316.715,Z 517.629,A -85,B 0,C 180,E1 -16140.405,E2 -16140.405} C_VEL
LIN {X 0,Y 312.357,Z 512.238,A -85,B 0,C 180,E1 -16141.32,E2 -16141.32} C_VEL
LIN {X 0,Y 308.79,Z 507.626,A -85,B 0,C 180,E1 -16142.028,E2 -16142.028} C_VEL
LIN {X 0,Y 307.438,Z 505.661,A -85,B 0,C 180,E1 -16142.294,E2 -16142.294} C_VEL
LIN {X 0,Y 305.857,Z 503.13,A -85,B 0,C 180,E1 -16142.625,E2 -16142.625} C_VEL
LIN {X 0,Y 305.501,Z 501.864,A -85,B 0,C 180,E1 -16142.869,E2 -16142.869} C_VEL
LIN {X 0,Y 305.459,Z 501.563,A -85,B 0,C 180,E1 -16144.078,E2 -16144.078} C_VEL
LIN {X 0,Y 305.492,Z 501.522,A -85,B 0,C 180,E1 -16146.736,E2 -16146.736} C_VEL
LIN {X 0,Y 305.489,Z 501.545,A -85,B 0,C 180,E1 -16150.608,E2 -16150.608} C_VEL
LIN {X 0,Y 305.538,Z 501.512,A -85,B 0,C 180,E1 -16154.516,E2 -16154.516} C_VEL
LIN {X 0,Y 305.495,Z 501.547,A -85,B 0,C 180,E1 -16158.153,E2 -16158.153} C_VEL
LIN {X 0,Y 305.511,Z 501.555,A -85,B 0,C 180,E1 -16161.604,E2 -16161.604} C_VEL
LIN {X 0,Y 305.455,Z 501.549,A -85,B 0,C 180,E1 -16164.887,E2 -16164.887} C_VEL
LIN {X 0,Y 305.448,Z 501.547,A -85,B 0,C 180,E1 -16168.354,E2 -16168.354} C_VEL
LIN {X 0,Y 305.514,Z 501.547,A -85,B 0,C 180,E1 -16171.114,E2 -16171.114} C_VEL
LIN {X 0,Y 305.564,Z 501.535,A -85,B 0,C 180,E1 -16174.088,E2 -16174.088} C_VEL
LIN {X 0,Y 305.493,Z 501.555,A -85,B 0,C 180,E1 -16178.403,E2 -16178.403} C_VEL
LIN {X 0,Y 305.582,Z 501.529,A -85,B 0,C 180,E1 -16181.218,E2 -16181.218} C_VEL
LIN {X 0,Y 305.641,Z 501.535,A -85,B 0,C 180,E1 -16185.349,E2 -16185.349} C_VEL
LIN {X 0,Y 305.628,Z 501.512,A -85,B 0,C 180,E1 -16189.4,E2 -16189.4} C_VEL
LIN {X 0,Y 305.79,Z 501.505,A -85,B 0,C 180,E1 -16192.074,E2 -16192.074} C_VEL
LIN {X 0,Y 305.683,Z 501.528,A -85,B 0,C 180,E1 -16194.724,E2 -16194.724} C_VEL
LIN {X 0,Y 305.95,Z 501.469,A -85,B 0,C 180,E1 -16198.684,E2 -16198.684} C_VEL
LIN {X 0,Y 305.95,Z 501.496,A -85,B 0,C 180,E1 -16201.317,E2 -16201.317} C_VEL
LIN {X 0,Y 305.89,Z 501.5,A -85,B 0,C 180,E1 -16202.075,E2 -16202.075} C_VEL
LIN {X 0,Y 305.185,Z 501.587,A -85,B 0,C 180,E1 -16203.172,E2 -16203.172} C_VEL
LIN {X 0,Y 302.283,Z 501.933,A -85,B 0,C 180,E1 -16204.957,E2 -16204.957} C_VEL
LIN {X 0,Y 299.849,Z 502.231,A -85,B 0,C 180,E1 -16206.405,E2 -16206.405} C_VEL
LIN {X 0,Y 298.82,Z 502.372,A -85,B 0,C 180,E1 -16207.528,E2 -16207.528} C_VEL
LIN {X 0,Y 298.744,Z 502.384,A -85,B 0,C 180,E1 -16207.908,E2 -16207.908} C_VEL
LIN {X 0,Y 298.587,Z 502.411,A -85,B 0,C 180,E1 -16210.854,E2 -16210.854} C_VEL
LIN {X 0,Y 298.58,Z 502.401,A -85,B 0,C 180,E1 -16215.195,E2 -16215.195} C_VEL
LIN {X 0,Y 298.52,Z 502.41,A -85,B 0,C 180,E1 -16219.245,E2 -16219.245} C_VEL
LIN {X 0,Y 298.424,Z 502.435,A -85,B 0,C 180,E1 -16223.601,E2 -16223.601} C_VEL
LIN {X 0,Y 298.48,Z 502.409,A -85,B 0,C 180,E1 -16226.576,E2 -16226.576} C_VEL
LIN {X 0,Y 298.413,Z 502.437,A -85,B 0,C 180,E1 -16229.642,E2 -16229.642} C_VEL
LIN {X 0,Y 298.391,Z 502.422,A -85,B 0,C 180,E1 -16232.801,E2 -16232.801} C_VEL
LIN {X 0,Y 298.463,Z 502.425,A -85,B 0,C 180,E1 -16236.814,E2 -16236.814} C_VEL
LIN {X 0,Y 298.415,Z 502.433,A -85,B 0,C 180,E1 -16241.095,E2 -16241.095} C_VEL
LIN {X 0,Y 298.424,Z 502.436,A -85,B 0,C 180,E1 -16243.11,E2 -16243.11} C_VEL
LIN {X 0,Y 298.402,Z 502.408,A -85,B 0,C 180,E1 -16246.922,E2 -16246.922} C_VEL
LIN {X 0,Y 298.44,Z 502.542,A -85,B 0,C 180,E1 -16250.411,E2 -16250.411} C_VEL
LIN {X 0,Y 300.655,Z 511.905,A -85,B 0,C 180,E1 -16254.241,E2 -16254.241} C_VEL
LIN {X 0,Y 302.088,Z 518.547,A -85,B 0,C 180,E1 -16256.763,E2 -16256.763} C_VEL
LIN {X 0,Y 303.902,Z 522.612,A -85,B 0,C 180,E1 -16257.165,E2 -16257.165} C_VEL
LIN {X 0,Y 311.915,Z 540.911,A -85,B 0,C 180,E1 -16258.587,E2 -16258.587} C_VEL
LIN {X 0,Y 316.785,Z 564.519,A -85,B 0,C 180,E1 -16259.727,E2 -16259.727} C_VEL
LIN {X 0,Y 317.86,Z 571.287,A -85,B 0,C 180,E1 -16260.012,E2 -16260.012} C_VEL
LIN {X 0,Y 315.225,Z 654.514,A -85,B 0,C 180,E1 -16261.902,E2 -16261.902} C_VEL
LIN {X 0,Y 314.46,Z 665.421,A -85,B 0,C 180,E1 -16262.281,E2 -16262.281} C_VEL
LIN {X 0,Y 313.435,Z 676.41,A -85,B 0,C 180,E1 -16262.816,E2 -16262.816} C_VEL
LIN {X 0,Y 312.279,Z 686.201,A -85,B 0,C 180,E1 -16263.43,E2 -16263.43} C_VEL
LIN {X 0,Y 310.953,Z 696.171,A -85,B 0,C 180,E1 -16264.21,E2 -16264.21} C_VEL
LIN {X 0,Y 309.316,Z 706.676,A -85,B 0,C 180,E1 -16265.216,E2 -16265.216} C_VEL
LIN {X 0,Y 307.87,Z 715.817,A -85,B 0,C 180,E1 -16266.276,E2 -16266.276} C_VEL
LIN {X 0,Y 306.138,Z 725.236,A -85,B 0,C 180,E1 -16267.564,E2 -16267.564} C_VEL
LIN {X 0,Y 304.255,Z 734.253,A -85,B 0,C 180,E1 -16269.021,E2 -16269.021} C_VEL
LIN {X 0,Y 302.885,Z 741.229,A -85,B 0,C 180,E1 -16270.34,E2 -16270.34} C_VEL
LIN {X 0,Y 301.338,Z 748.753,A -85,B 0,C 180,E1 -16272,E2 -16272} C_VEL
LIN {X 0,Y 299.864,Z 756.097,A -85,B 0,C 180,E1 -16273.933,E2 -16273.933} C_VEL
LIN {X 0,Y 298.901,Z 761.774,A -85,B 0,C 180,E1 -16275.707,E2 -16275.707} C_VEL
LIN {X 0,Y 297.886,Z 767.207,A -85,B 0,C 180,E1 -16277.741,E2 -16277.741} C_VEL
LIN {X 0,Y 297.223,Z 771.655,A -85,B 0,C 180,E1 -16279.785,E2 -16279.785} C_VEL
LIN {X 0,Y 296.824,Z 775.203,A -85,B 0,C 180,E1 -16281.833,E2 -16281.833} C_VEL
LIN {X 0,Y 296.646,Z 777.145,A -85,B 0,C 180,E1 -16283.197,E2 -16283.197} C_VEL
LIN {X 0,Y 296.487,Z 779.833,A -85,B 0,C 180,E1 -16285.922,E2 -16285.922} C_VEL
LIN {X 0,Y 296.524,Z 780.653,A -85,B 0,C 180,E1 -16287.283,E2 -16287.283} C_VEL
LIN {X 0,Y 296.519,Z 781.379,A -85,B 0,C 180,E1 -16290,E2 -16290} C_VEL
LIN {X 0,Y 296.524,Z 780.653,A -85,B 0,C 180,E1 -16292.717,E2 -16292.717} C_VEL
LIN {X 0,Y 296.488,Z 779.833,A -85,B 0,C 180,E1 -16294.078,E2 -16294.078} C_VEL
LIN {X 0,Y 296.646,Z 777.145,A -85,B 0,C 180,E1 -16296.803,E2 -16296.803} C_VEL
LIN {X 0,Y 296.944,Z 774.187,A -85,B 0,C 180,E1 -16298.849,E2 -16298.849} C_VEL
LIN {X 0,Y 297.396,Z 770.356,A -85,B 0,C 180,E1 -16300.897,E2 -16300.897} C_VEL
LIN {X 0,Y 298.242,Z 765.593,A -85,B 0,C 180,E1 -16302.936,E2 -16302.936} C_VEL
LIN {X 0,Y 299.53,Z 758.437,A -85,B 0,C 180,E1 -16305.369,E2 -16305.369} C_VEL
LIN {X 0,Y 300.794,Z 751.429,A -85,B 0,C 180,E1 -16307.331,E2 -16307.331} C_VEL
LIN {X 0,Y 302.237,Z 744.353,A -85,B 0,C 180,E1 -16308.998,E2 -16308.998} C_VEL
LIN {X 0,Y 303.887,Z 736.072,A -85,B 0,C 180,E1 -16310.651,E2 -16310.651} C_VEL
LIN {X 0,Y 305.69,Z 727.354,A -85,B 0,C 180,E1 -16312.115,E2 -16312.115} C_VEL
LIN {X 0,Y 307.491,Z 718.299,A -85,B 0,C 180,E1 -16313.398,E2 -16313.398} C_VEL
LIN {X 0,Y 308.942,Z 709.247,A -85,B 0,C 180,E1 -16314.501,E2 -16314.501} C_VEL
LIN {X 0,Y 310.424,Z 699.678,A -85,B 0,C 180,E1 -16315.477,E2 -16315.477} C_VEL
LIN {X 0,Y 311.829,Z 689.42,A -85,B 0,C 180,E1 -16316.341,E2 -16316.341} C_VEL
LIN {X 0,Y 313.268,Z 677.769,A -85,B 0,C 180,E1 -16317.109,E2 -16317.109} C_VEL
LIN {X 0,Y 314.376,Z 666.332,A -85,B 0,C 180,E1 -16317.682,E2 -16317.682} C_VEL
LIN {X 0,Y 315.125,Z 655.83,A -85,B 0,C 180,E1 -16318.062,E2 -16318.062} C_VEL
LIN {X 0,Y 316.205,Z 625.719,A -85,B 0,C 180,E1 -16318.772,E2 -16318.772} C_VEL
LIN {X 0,Y 317.821,Z 570.147,A -85,B 0,C 180,E1 -16320.021,E2 -16320.021} C_VEL
LIN {X 0,Y 312.929,Z 545.277,A -85,B 0,C 180,E1 -16321.186,E2 -16321.186} C_VEL
LIN {X 0,Y 311.441,Z 539.675,A -85,B 0,C 180,E1 -16321.499,E2 -16321.499} C_VEL
LIN {X 0,Y 303.77,Z 522.383,A -85,B 0,C 180,E1 -16322.857,E2 -16322.857} C_VEL
LIN {X 0,Y 302.061,Z 518.581,A -85,B 0,C 180,E1 -16323.23,E2 -16323.23} C_VEL
LIN {X 0,Y 300.658,Z 511.905,A -85,B 0,C 180,E1 -16325.759,E2 -16325.759} C_VEL
LIN {X 0,Y 298.428,Z 502.45,A -85,B 0,C 180,E1 -16329.673,E2 -16329.673} C_VEL
LIN {X 0,Y 298.397,Z 502.408,A -85,B 0,C 180,E1 -16333.102,E2 -16333.102} C_VEL
LIN {X 0,Y 298.43,Z 502.433,A -85,B 0,C 180,E1 -16336.925,E2 -16336.925} C_VEL
LIN {X 0,Y 298.423,Z 502.429,A -85,B 0,C 180,E1 -16341,E2 -16341} C_VEL
LIN {X 0,Y 298.429,Z 502.437,A -85,B 0,C 180,E1 -16343.931,E2 -16343.931} C_VEL
LIN {X 0,Y 298.389,Z 502.428,A -85,B 0,C 180,E1 -16347.983,E2 -16347.983} C_VEL
LIN {X 0,Y 298.444,Z 502.416,A -85,B 0,C 180,E1 -16351.902,E2 -16351.902} C_VEL
LIN {X 0,Y 298.477,Z 502.425,A -85,B 0,C 180,E1 -16354.923,E2 -16354.923} C_VEL
LIN {X 0,Y 298.431,Z 502.41,A -85,B 0,C 180,E1 -16359.313,E2 -16359.313} C_VEL
LIN {X 0,Y 298.529,Z 502.422,A -85,B 0,C 180,E1 -16362.178,E2 -16362.178} C_VEL
LIN {X 0,Y 298.587,Z 502.397,A -85,B 0,C 180,E1 -16364.994,E2 -16364.994} C_VEL
LIN {X 0,Y 298.587,Z 502.411,A -85,B 0,C 180,E1 -16369.146,E2 -16369.146} C_VEL
LIN {X 0,Y 298.749,Z 502.387,A -85,B 0,C 180,E1 -16371.885,E2 -16371.885} C_VEL
LIN {X 0,Y 298.652,Z 502.374,A -85,B 0,C 180,E1 -16374.598,E2 -16374.598} C_VEL
LIN {X 0,Y 298.917,Z 502.372,A -85,B 0,C 180,E1 -16378.652,E2 -16378.652} C_VEL
LIN {X 0,Y 298.917,Z 502.344,A -85,B 0,C 180,E1 -16381.347,E2 -16381.347} C_VEL
LIN {X 0,Y 298.78,Z 502.389,A -85,B 0,C 180,E1 -16386.754,E2 -16386.754} C_VEL
LIN {X 0,Y 298.628,Z 502.381,A -85,B 0,C 180,E1 -16389.481,E2 -16389.481} C_VEL
LIN {X 0,Y 298.545,Z 502.424,A -85,B 0,C 180,E1 -16393.615,E2 -16393.615} C_VEL
LIN {X 0,Y 298.541,Z 502.4,A -85,B 0,C 180,E1 -16396.408,E2 -16396.408} C_VEL
LIN {X 0,Y 298.504,Z 502.419,A -85,B 0,C 180,E1 -16399.654,E2 -16399.654} C_VEL
LIN {X 0,Y 298.45,Z 502.411,A -85,B 0,C 180,E1 -16403.597,E2 -16403.597} C_VEL
LIN {X 0,Y 298.483,Z 502.427,A -85,B 0,C 180,E1 -16406.574,E2 -16406.574} C_VEL
LIN {X 0,Y 298.415,Z 502.42,A -85,B 0,C 180,E1 -16409.641,E2 -16409.641} C_VEL
LIN {X 0,Y 298.39,Z 502.44,A -85,B 0,C 180,E1 -16412.8,E2 -16412.8} C_VEL
LIN {X 0,Y 298.459,Z 502.42,A -85,B 0,C 180,E1 -16416.812,E2 -16416.812} C_VEL
LIN {X 0,Y 298.447,Z 502.42,A -85,B 0,C 180,E1 -16421.102,E2 -16421.102} C_VEL
LIN {X 0,Y 298.483,Z 502.398,A -85,B 0,C 180,E1 -16425.061,E2 -16425.061} C_VEL
LIN {X 0,Y 298.45,Z 502.407,A -85,B 0,C 180,E1 -16428.897,E2 -16428.897} C_VEL
LIN {X 0,Y 298.46,Z 502.397,A -85,B 0,C 180,E1 -16433.188,E2 -16433.188} C_VEL
LIN {X 0,Y 298.462,Z 502.661,A -85,B 0,C 180,E1 -16436.111,E2 -16436.111} C_VEL
LIN {X 0,Y 298.669,Z 503.583,A -85,B 0,C 180,E1 -16436.354,E2 -16436.354} C_VEL
LIN {X 0,Y 300.334,Z 506.514,A -85,B 0,C 180,E1 -16436.703,E2 -16436.703} C_VEL
LIN {X 0,Y 303.493,Z 511.091,A -85,B 0,C 180,E1 -16437.267,E2 -16437.267} C_VEL
LIN {X 0,Y 307.12,Z 516.032,A -85,B 0,C 180,E1 -16437.968,E2 -16437.968} C_VEL
LIN {X 0,Y 311.58,Z 521.404,A -85,B 0,C 180,E1 -16438.833,E2 -16438.833} C_VEL
LIN {X 0,Y 316.6,Z 527.161,A -85,B 0,C 180,E1 -16439.876,E2 -16439.876} C_VEL
LIN {X 0,Y 321.913,Z 533.006,A -85,B 0,C 180,E1 -16441.071,E2 -16441.071} C_VEL
LIN {X 0,Y 326.729,Z 538.411,A -85,B 0,C 180,E1 -16442.236,E2 -16442.236} C_VEL
LIN {X 0,Y 332.872,Z 544.803,A -85,B 0,C 180,E1 -16443.773,E2 -16443.773} C_VEL
LIN {X 0,Y 338.92,Z 550.898,A -85,B 0,C 180,E1 -16445.376,E2 -16445.376} C_VEL
LIN {X 0,Y 341.906,Z 553.732,A -85,B 0,C 180,E1 -16446.201,E2 -16446.201} C_VEL
LIN {X 0,Y 346.394,Z 557.958,A -85,B 0,C 180,E1 -16447.494,E2 -16447.494} C_VEL
LIN {X 0,Y 349.95,Z 561.31,A -85,B 0,C 180,E1 -16448.578,E2 -16448.578} C_VEL
LIN {X 0,Y 354.593,Z 565.318,A -85,B 0,C 180,E1 -16450.054,E2 -16450.054} C_VEL
LIN {X 0,Y 356.686,Z 567.153,A -85,B 0,C 180,E1 -16450.762,E2 -16450.762} C_VEL
LIN {X 0,Y 361.028,Z 571.171,A -85,B 0,C 180,E1 -16452.329,E2 -16452.329} C_VEL
LIN {X 0,Y 364.933,Z 574.089,A -85,B 0,C 180,E1 -16453.828,E2 -16453.828} C_VEL
LIN {X 0,Y 368.951,Z 577.914,A -85,B 0,C 180,E1 -16455.574,E2 -16455.574} C_VEL
LIN {X 0,Y 372.503,Z 580.346,A -85,B 0,C 180,E1 -16457.263,E2 -16457.263} C_VEL
LIN {X 0,Y 374.673,Z 581.746,A -85,B 0,C 180,E1 -16458.405,E2 -16458.405} C_VEL
LIN {X 0,Y 377.94,Z 585.022,A -85,B 0,C 180,E1 -16460.482,E2 -16460.482} C_VEL
LIN {X 0,Y 380.38,Z 586.8,A -85,B 0,C 180,E1 -16462.327,E2 -16462.327} C_VEL
LIN {X 0,Y 382.595,Z 588.06,A -85,B 0,C 180,E1 -16464.446,E2 -16464.446} C_VEL
LIN {X 0,Y 383.631,Z 588.512,A -85,B 0,C 180,E1 -16465.798,E2 -16465.798} C_VEL
LIN {X 0,Y 384.717,Z 588.927,A -85,B 0,C 180,E1 -16467.906,E2 -16467.906} C_VEL
LIN {X 0,Y 384.977,Z 589.128,A -85,B 0,C 180,E1 -16468.954,E2 -16468.954} C_VEL
LIN {X 0,Y 385.084,Z 589.021,A -85,B 0,C 180,E1 -16470,E2 -16470} C_VEL
LIN {X 0,Y 384.976,Z 589.13,A -85,B 0,C 180,E1 -16471.046,E2 -16471.046} C_VEL
LIN {X 0,Y 384.277,Z 588.656,A -85,B 0,C 180,E1 -16473.145,E2 -16473.145} C_VEL
LIN {X 0,Y 382.835,Z 588.164,A -85,B 0,C 180,E1 -16475.266,E2 -16475.266} C_VEL
LIN {X 0,Y 380.681,Z 586.946,A -85,B 0,C 180,E1 -16477.425,E2 -16477.425} C_VEL
LIN {X 0,Y 378.008,Z 585.091,A -85,B 0,C 180,E1 -16479.47,E2 -16479.47} C_VEL
LIN {X 0,Y 374.802,Z 581.915,A -85,B 0,C 180,E1 -16481.515,E2 -16481.515} C_VEL
LIN {X 0,Y 373.355,Z 580.804,A -85,B 0,C 180,E1 -16482.303,E2 -16482.303} C_VEL
LIN {X 0,Y 369.596,Z 578.417,A -85,B 0,C 180,E1 -16484.124,E2 -16484.124} C_VEL
LIN {X 0,Y 365.696,Z 574.893,A -85,B 0,C 180,E1 -16485.848,E2 -16485.848} C_VEL
LIN {X 0,Y 363.596,Z 572.981,A -85,B 0,C 180,E1 -16486.705,E2 -16486.705} C_VEL
LIN {X 0,Y 359.246,Z 569.663,A -85,B 0,C 180,E1 -16488.326,E2 -16488.326} C_VEL
LIN {X 0,Y 354.826,Z 565.467,A -85,B 0,C 180,E1 -16489.869,E2 -16489.869} C_VEL
LIN {X 0,Y 350.28,Z 561.639,A -85,B 0,C 180,E1 -16491.318,E2 -16491.318} C_VEL
LIN {X 0,Y 346.856,Z 558.331,A -85,B 0,C 180,E1 -16492.368,E2 -16492.368} C_VEL
LIN {X 0,Y 342.288,Z 554.139,A -85,B 0,C 180,E1 -16493.69,E2 -16493.69} C_VEL
LIN {X 0,Y 338.304,Z 550.354,A -85,B 0,C 180,E1 -16494.786,E2 -16494.786} C_VEL
LIN {X 0,Y 331.831,Z 543.83,A -85,B 0,C 180,E1 -16496.488,E2 -16496.488} C_VEL
LIN {X 0,Y 323.311,Z 534.721,A -85,B 0,C 180,E1 -16498.592,E2 -16498.592} C_VEL
LIN {X 0,Y 317.676,Z 528.273,A -85,B 0,C 180,E1 -16499.89,E2 -16499.89} C_VEL
LIN {X 0,Y 313.266,Z 523.438,A -85,B 0,C 180,E1 -16500.819,E2 -16500.819} C_VEL
LIN {X 0,Y 308.3,Z 517.452,A -85,B 0,C 180,E1 -16501.812,E2 -16501.812} C_VEL
LIN {X 0,Y 304.345,Z 512.335,A -85,B 0,C 180,E1 -16502.573,E2 -16502.573} C_VEL
LIN {X 0,Y 301.116,Z 507.706,A -85,B 0,C 180,E1 -16503.156,E2 -16503.156} C_VEL
LIN {X 0,Y 298.829,Z 504.034,A -85,B 0,C 180,E1 -16503.594,E2 -16503.594} C_VEL
LIN {X 0,Y 298.483,Z 502.764,A -85,B 0,C 180,E1 -16503.837,E2 -16503.837} C_VEL
LIN {X 0,Y 298.423,Z 502.43,A -85,B 0,C 180,E1 -16504.487,E2 -16504.487} C_VEL
LIN {X 0,Y 298.435,Z 502.406,A -85,B 0,C 180,E1 -16507.754,E2 -16507.754} C_VEL
LIN {X 0,Y 298.451,Z 502.403,A -85,B 0,C 180,E1 -16511.249,E2 -16511.249} C_VEL
LIN {X 0,Y 298.483,Z 502.4,A -85,B 0,C 180,E1 -16515.061,E2 -16515.061} C_VEL
LIN {X 0,Y 298.447,Z 502.42,A -85,B 0,C 180,E1 -16518.898,E2 -16518.898} C_VEL
LIN {X 0,Y 298.459,Z 502.42,A -85,B 0,C 180,E1 -16523.188,E2 -16523.188} C_VEL
LIN {X 0,Y 298.39,Z 502.44,A -85,B 0,C 180,E1 -16527.2,E2 -16527.2} C_VEL
LIN {X 0,Y 298.426,Z 502.421,A -85,B 0,C 180,E1 -16530.615,E2 -16530.615} C_VEL
LIN {X 0,Y 298.477,Z 502.428,A -85,B 0,C 180,E1 -16533.474,E2 -16533.474} C_VEL
LIN {X 0,Y 298.427,Z 502.416,A -85,B 0,C 180,E1 -16536.698,E2 -16536.698} C_VEL
LIN {X 0,Y 298.532,Z 502.412,A -85,B 0,C 180,E1 -16540.757,E2 -16540.757} C_VEL
LIN {X 0,Y 298.586,Z 502.412,A -85,B 0,C 180,E1 -16544.995,E2 -16544.995} C_VEL
LIN {X 0,Y 298.584,Z 502.391,A -85,B 0,C 180,E1 -16549.147,E2 -16549.147} C_VEL
LIN {X 0,Y 298.735,Z 502.382,A -85,B 0,C 180,E1 -16551.886,E2 -16551.886} C_VEL
LIN {X 0,Y 298.653,Z 502.404,A -85,B 0,C 180,E1 -16554.599,E2 -16554.599} C_VEL
LIN {X 0,Y 298.917,Z 502.344,A -85,B 0,C 180,E1 -16558.653,E2 -16558.653} C_VEL
LIN {X 0,Y 298.917,Z 502.372,A -85,B 0,C 180,E1 -16561.348,E2 -16561.348} C_VEL
LIN {X 0,Y 298.786,Z 502.363,A -85,B 0,C 180,E1 -16566.755,E2 -16566.755} C_VEL
LIN {X 0,Y 298.744,Z 502.384,A -85,B 0,C 180,E1 -16567.908,E2 -16567.908} C_VEL
LIN {X 0,Y 298.065,Z 502.482,A -85,B 0,C 180,E1 -16569.032,E2 -16569.032} C_VEL
LIN {X 0,Y 295.105,Z 502.844,A -85,B 0,C 180,E1 -16570.858,E2 -16570.858} C_VEL
LIN {X 0,Y 292.61,Z 503.136,A -85,B 0,C 180,E1 -16572.34,E2 -16572.34} C_VEL
LIN {X 0,Y 291.575,Z 503.258,A -85,B 0,C 180,E1 -16573.491,E2 -16573.491} C_VEL
LIN {X 0,Y 291.511,Z 503.266,A -85,B 0,C 180,E1 -16573.881,E2 -16573.881} C_VEL
LIN {X 0,Y 291.481,Z 503.303,A -85,B 0,C 180,E1 -16576.819,E2 -16576.819} C_VEL
LIN {X 0,Y 291.446,Z 503.282,A -85,B 0,C 180,E1 -16579.876,E2 -16579.876} C_VEL
LIN {X 0,Y 291.378,Z 503.315,A -85,B 0,C 180,E1 -16584.208,E2 -16584.208} C_VEL
LIN {X 0,Y 291.411,Z 503.287,A -85,B 0,C 180,E1 -16587.273,E2 -16587.273} C_VEL
LIN {X 0,Y 291.33,Z 503.323,A -85,B 0,C 180,E1 -16590.438,E2 -16590.438} C_VEL
LIN {X 0,Y 291.341,Z 503.302,A -85,B 0,C 180,E1 -16593.699,E2 -16593.699} C_VEL
LIN {X 0,Y 291.395,Z 503.301,A -85,B 0,C 180,E1 -16597.261,E2 -16597.261} C_VEL
LIN {X 0,Y 291.374,Z 503.315,A -85,B 0,C 180,E1 -16600.636,E2 -16600.636} C_VEL
LIN {X 0,Y 291.298,Z 503.321,A -85,B 0,C 180,E1 -16604.401,E2 -16604.401} C_VEL
LIN {X 0,Y 291.325,Z 503.304,A -85,B 0,C 180,E1 -16608.405,E2 -16608.405} C_VEL
LIN {X 0,Y 291.413,Z 503.521,A -85,B 0,C 180,E1 -16609.77,E2 -16609.77} C_VEL
LIN {X 0,Y 293.343,Z 511.652,A -85,B 0,C 180,E1 -16613.206,E2 -16613.206} C_VEL
LIN {X 0,Y 294.883,Z 518.416,A -85,B 0,C 180,E1 -16615.861,E2 -16615.861} C_VEL
LIN {X 0,Y 299.92,Z 529.368,A -85,B 0,C 180,E1 -16616.866,E2 -16616.866} C_VEL
LIN {X 0,Y 306.2,Z 543.933,A -85,B 0,C 180,E1 -16618.018,E2 -16618.018} C_VEL
LIN {X 0,Y 310.759,Z 566.319,A -85,B 0,C 180,E1 -16619.129,E2 -16619.129} C_VEL
LIN {X 0,Y 311.714,Z 571.812,A -85,B 0,C 180,E1 -16619.377,E2 -16619.377} C_VEL
LIN {X 0,Y 308.976,Z 654.323,A -85,B 0,C 180,E1 -16621.282,E2 -16621.282} C_VEL
LIN {X 0,Y 308.206,Z 665.223,A -85,B 0,C 180,E1 -16621.668,E2 -16621.668} C_VEL
LIN {X 0,Y 307.141,Z 676.212,A -85,B 0,C 180,E1 -16622.211,E2 -16622.211} C_VEL
LIN {X 0,Y 305.925,Z 686.002,A -85,B 0,C 180,E1 -16622.834,E2 -16622.834} C_VEL
LIN {X 0,Y 304.557,Z 695.973,A -85,B 0,C 180,E1 -16623.628,E2 -16623.628} C_VEL
LIN {X 0,Y 302.872,Z 706.477,A -85,B 0,C 180,E1 -16624.652,E2 -16624.652} C_VEL
LIN {X 0,Y 301.437,Z 715.212,A -85,B 0,C 180,E1 -16625.678,E2 -16625.678} C_VEL
LIN {X 0,Y 299.527,Z 725.036,A -85,B 0,C 180,E1 -16627.041,E2 -16627.041} C_VEL
LIN {X 0,Y 297.619,Z 734.055,A -85,B 0,C 180,E1 -16628.53,E2 -16628.53} C_VEL
LIN {X 0,Y 296.157,Z 741.03,A -85,B 0,C 180,E1 -16629.874,E2 -16629.874} C_VEL
LIN {X 0,Y 294.56,Z 748.554,A -85,B 0,C 180,E1 -16631.571,E2 -16631.571} C_VEL
LIN {X 0,Y 293.194,Z 755.029,A -85,B 0,C 180,E1 -16633.283,E2 -16633.283} C_VEL
LIN {X 0,Y 291.97,Z 761.575,A -85,B 0,C 180,E1 -16635.36,E2 -16635.36} C_VEL
LIN {X 0,Y 290.925,Z 767.009,A -85,B 0,C 180,E1 -16637.443,E2 -16637.443} C_VEL
LIN {X 0,Y 290.178,Z 771.455,A -85,B 0,C 180,E1 -16639.535,E2 -16639.535} C_VEL
LIN {X 0,Y 289.76,Z 775.004,A -85,B 0,C 180,E1 -16641.632,E2 -16641.632} C_VEL
LIN {X 0,Y 289.571,Z 776.947,A -85,B 0,C 180,E1 -16643.03,E2 -16643.03} C_VEL
LIN {X 0,Y 289.393,Z 779.634,A -85,B 0,C 180,E1 -16645.822,E2 -16645.822} C_VEL
LIN {X 0,Y 289.427,Z 780.455,A -85,B 0,C 180,E1 -16647.216,E2 -16647.216} C_VEL
LIN {X 0,Y 289.436,Z 781.181,A -85,B 0,C 180,E1 -16650,E2 -16650} C_VEL
LIN {X 0,Y 289.427,Z 780.455,A -85,B 0,C 180,E1 -16652.784,E2 -16652.784} C_VEL
LIN {X 0,Y 289.434,Z 778.573,A -85,B 0,C 180,E1 -16655.399,E2 -16655.399} C_VEL
LIN {X 0,Y 289.571,Z 776.947,A -85,B 0,C 180,E1 -16656.97,E2 -16656.97} C_VEL
LIN {X 0,Y 289.882,Z 773.987,A -85,B 0,C 180,E1 -16659.067,E2 -16659.067} C_VEL
LIN {X 0,Y 290.365,Z 770.156,A -85,B 0,C 180,E1 -16661.165,E2 -16661.165} C_VEL
LIN {X 0,Y 291.268,Z 765.393,A -85,B 0,C 180,E1 -16663.251,E2 -16663.251} C_VEL
LIN {X 0,Y 292.567,Z 758.514,A -85,B 0,C 180,E1 -16665.657,E2 -16665.657} C_VEL
LIN {X 0,Y 293.685,Z 752.567,A -85,B 0,C 180,E1 -16667.405,E2 -16667.405} C_VEL
LIN {X 0,Y 295.485,Z 744.154,A -85,B 0,C 180,E1 -16669.45,E2 -16669.45} C_VEL
LIN {X 0,Y 297.202,Z 735.872,A -85,B 0,C 180,E1 -16671.138,E2 -16671.138} C_VEL
LIN {X 0,Y 299.112,Z 727.155,A -85,B 0,C 180,E1 -16672.628,E2 -16672.628} C_VEL
LIN {X 0,Y 300.964,Z 718.138,A -85,B 0,C 180,E1 -16673.931,E2 -16673.931} C_VEL
LIN {X 0,Y 302.458,Z 709.117,A -85,B 0,C 180,E1 -16675.054,E2 -16675.054} C_VEL
LIN {X 0,Y 304.015,Z 699.48,A -85,B 0,C 180,E1 -16676.054,E2 -16676.054} C_VEL
LIN {X 0,Y 305.47,Z 689.222,A -85,B 0,C 180,E1 -16676.933,E2 -16676.933} C_VEL
LIN {X 0,Y 306.98,Z 677.571,A -85,B 0,C 180,E1 -16677.712,E2 -16677.712} C_VEL
LIN {X 0,Y 308.107,Z 666.134,A -85,B 0,C 180,E1 -16678.295,E2 -16678.295} C_VEL
LIN {X 0,Y 308.884,Z 655.633,A -85,B 0,C 180,E1 -16678.681,E2 -16678.681} C_VEL
LIN {X 0,Y 310.004,Z 625.521,A -85,B 0,C 180,E1 -16679.403,E2 -16679.403} C_VEL
LIN {X 0,Y 311.603,Z 571.213,A -85,B 0,C 180,E1 -16680.651,E2 -16680.651} C_VEL
LIN {X 0,Y 307.458,Z 549.408,A -85,B 0,C 180,E1 -16681.69,E2 -16681.69} C_VEL
LIN {X 0,Y 305.726,Z 542.562,A -85,B 0,C 180,E1 -16682.074,E2 -16682.074} C_VEL
LIN {X 0,Y 298.383,Z 526.055,A -85,B 0,C 180,E1 -16683.419,E2 -16683.419} C_VEL
LIN {X 0,Y 294.974,Z 518.6,A -85,B 0,C 180,E1 -16684.102,E2 -16684.102} C_VEL
LIN {X 0,Y 294.369,Z 516.141,A -85,B 0,C 180,E1 -16684.958,E2 -16684.958} C_VEL
LIN {X 0,Y 292.667,Z 508.672,A -85,B 0,C 180,E1 -16688.026,E2 -16688.026} C_VEL
LIN {X 0,Y 291.383,Z 503.329,A -85,B 0,C 180,E1 -16690.396,E2 -16690.396} C_VEL
LIN {X 0,Y 291.288,Z 503.299,A -85,B 0,C 180,E1 -16694.401,E2 -16694.401} C_VEL
LIN {X 0,Y 291.353,Z 503.308,A -85,B 0,C 180,E1 -16698.397,E2 -16698.397} C_VEL
LIN {X 0,Y 291.372,Z 503.305,A -85,B 0,C 180,E1 -16701.161,E2 -16701.161} C_VEL
LIN {X 0,Y 291.383,Z 503.315,A -85,B 0,C 180,E1 -16704.628,E2 -16704.628} C_VEL
LIN {X 0,Y 291.366,Z 503.302,A -85,B 0,C 180,E1 -16707.949,E2 -16707.949} C_VEL
LIN {X 0,Y 291.369,Z 503.305,A -85,B 0,C 180,E1 -16711.156,E2 -16711.156} C_VEL
LIN {X 0,Y 291.407,Z 503.299,A -85,B 0,C 180,E1 -16714.27,E2 -16714.27} C_VEL
LIN {X 0,Y 291.369,Z 503.306,A -85,B 0,C 180,E1 -16717.298,E2 -16717.298} C_VEL
LIN {X 0,Y 291.453,Z 503.283,A -85,B 0,C 180,E1 -16720.269,E2 -16720.269} C_VEL
LIN {X 0,Y 291.535,Z 503.281,A -85,B 0,C 180,E1 -16724.634,E2 -16724.634} C_VEL
LIN {X 0,Y 291.53,Z 503.288,A -85,B 0,C 180,E1 -16728.88,E2 -16728.88} C_VEL
LIN {X 0,Y 291.7,Z 503.267,A -85,B 0,C 180,E1 -16731.688,E2 -16731.688} C_VEL
LIN {X 0,Y 291.622,Z 503.249,A -85,B 0,C 180,E1 -16734.468,E2 -16734.468} C_VEL
LIN {X 0,Y 291.883,Z 503.248,A -85,B 0,C 180,E1 -16738.62,E2 -16738.62} C_VEL
LIN {X 0,Y 291.883,Z 503.219,A -85,B 0,C 180,E1 -16741.379,E2 -16741.379} C_VEL
LIN {X 0,Y 291.728,Z 503.268,A -85,B 0,C 180,E1 -16746.918,E2 -16746.918} C_VEL
LIN {X 0,Y 291.568,Z 503.259,A -85,B 0,C 180,E1 -16749.713,E2 -16749.713} C_VEL
LIN {X 0,Y 291.515,Z 503.298,A -85,B 0,C 180,E1 -16753.95,E2 -16753.95} C_VEL
LIN {X 0,Y 291.479,Z 503.275,A -85,B 0,C 180,E1 -16756.818,E2 -16756.818} C_VEL
LIN {X 0,Y 291.444,Z 503.301,A -85,B 0,C 180,E1 -16759.875,E2 -16759.875} C_VEL
LIN {X 0,Y 291.393,Z 503.286,A -85,B 0,C 180,E1 -16764.205,E2 -16764.205} C_VEL
LIN {X 0,Y 291.416,Z 503.309,A -85,B 0,C 180,E1 -16767.271,E2 -16767.271} C_VEL
LIN {X 0,Y 291.332,Z 503.297,A -85,B 0,C 180,E1 -16770.437,E2 -16770.437} C_VEL
LIN {X 0,Y 291.339,Z 503.32,A -85,B 0,C 180,E1 -16773.698,E2 -16773.698} C_VEL
LIN {X 0,Y 291.394,Z 503.304,A -85,B 0,C 180,E1 -16777.26,E2 -16777.26} C_VEL
LIN {X 0,Y 291.396,Z 503.297,A -85,B 0,C 180,E1 -16780.631,E2 -16780.631} C_VEL
LIN {X 0,Y 291.401,Z 503.294,A -85,B 0,C 180,E1 -16784.379,E2 -16784.379} C_VEL
LIN {X 0,Y 291.384,Z 503.275,A -85,B 0,C 180,E1 -16788.39,E2 -16788.39} C_VEL
LIN {X 0,Y 291.376,Z 503.303,A -85,B 0,C 180,E1 -16791.163,E2 -16791.163} C_VEL
LIN {X 0,Y 291.38,Z 503.288,A -85,B 0,C 180,E1 -16794.63,E2 -16794.63} C_VEL
LIN {X 0,Y 291.412,Z 503.573,A -85,B 0,C 180,E1 -16795.221,E2 -16795.221} C_VEL
LIN {X 0,Y 291.623,Z 504.482,A -85,B 0,C 180,E1 -16795.442,E2 -16795.442} C_VEL
LIN {X 0,Y 293.23,Z 507.309,A -85,B 0,C 180,E1 -16795.768,E2 -16795.768} C_VEL
LIN {X 0,Y 296.017,Z 511.644,A -85,B 0,C 180,E1 -16796.261,E2 -16796.261} C_VEL
LIN {X 0,Y 299.085,Z 516.132,A -85,B 0,C 180,E1 -16796.809,E2 -16796.809} C_VEL
LIN {X 0,Y 303.159,Z 521.438,A -85,B 0,C 180,E1 -16797.524,E2 -16797.524} C_VEL
LIN {X 0,Y 308.049,Z 527.187,A -85,B 0,C 180,E1 -16798.441,E2 -16798.441} C_VEL
LIN {X 0,Y 312.862,Z 532.646,A -85,B 0,C 180,E1 -16799.4,E2 -16799.4} C_VEL
LIN {X 0,Y 318.411,Z 538.616,A -85,B 0,C 180,E1 -16800.585,E2 -16800.585} C_VEL
LIN {X 0,Y 323.809,Z 544.458,A -85,B 0,C 180,E1 -16801.829,E2 -16801.829} C_VEL
LIN {X 0,Y 330.142,Z 550.984,A -85,B 0,C 180,E1 -16803.39,E2 -16803.39} C_VEL
LIN {X 0,Y 336.452,Z 557.23,A -85,B 0,C 180,E1 -16805.024,E2 -16805.024} C_VEL
LIN {X 0,Y 339.615,Z 560.224,A -85,B 0,C 180,E1 -16805.879,E2 -16805.879} C_VEL
LIN {X 0,Y 344.458,Z 564.623,A -85,B 0,C 180,E1 -16807.246,E2 -16807.246} C_VEL
LIN {X 0,Y 350.845,Z 570.489,A -85,B 0,C 180,E1 -16809.183,E2 -16809.183} C_VEL
LIN {X 0,Y 354.639,Z 573.602,A -85,B 0,C 180,E1 -16810.416,E2 -16810.416} C_VEL
LIN {X 0,Y 359.159,Z 577.713,A -85,B 0,C 180,E1 -16812.004,E2 -16812.004} C_VEL
LIN {X 0,Y 363.692,Z 581.164,A -85,B 0,C 180,E1 -16813.716,E2 -16813.716} C_VEL
LIN {X 0,Y 367.693,Z 584.859,A -85,B 0,C 180,E1 -16815.434,E2 -16815.434} C_VEL
LIN {X 0,Y 371.515,Z 587.359,A -85,B 0,C 180,E1 -16817.229,E2 -16817.229} C_VEL
LIN {X 0,Y 373.521,Z 588.761,A -85,B 0,C 180,E1 -16818.282,E2 -16818.282} C_VEL
LIN {X 0,Y 376.825,Z 591.968,A -85,B 0,C 180,E1 -16820.337,E2 -16820.337} C_VEL
LIN {X 0,Y 379.475,Z 593.851,A -85,B 0,C 180,E1 -16822.309,E2 -16822.309} C_VEL
LIN {X 0,Y 381.711,Z 595.104,A -85,B 0,C 180,E1 -16824.433,E2 -16824.433} C_VEL
LIN {X 0,Y 382.754,Z 595.556,A -85,B 0,C 180,E1 -16825.788,E2 -16825.788} C_VEL
LIN {X 0,Y 383.85,Z 595.968,A -85,B 0,C 180,E1 -16827.901,E2 -16827.901} C_VEL
LIN {X 0,Y 384.111,Z 596.174,A -85,B 0,C 180,E1 -16828.952,E2 -16828.952} C_VEL
LIN {X 0,Y 384.219,Z 596.068,A -85,B 0,C 180,E1 -16830,E2 -16830} C_VEL
LIN {X 0,Y 383.991,Z 596.082,A -85,B 0,C 180,E1 -16831.573,E2 -16831.573} C_VEL
LIN {X 0,Y 383.405,Z 595.704,A -85,B 0,C 180,E1 -16833.152,E2 -16833.152} C_VEL
LIN {X 0,Y 381.95,Z 595.211,A -85,B 0,C 180,E1 -16835.279,E2 -16835.279} C_VEL
LIN {X 0,Y 379.773,Z 594.015,A -85,B 0,C 180,E1 -16837.443,E2 -16837.443} C_VEL
LIN {X 0,Y 377.102,Z 592.149,A -85,B 0,C 180,E1 -16839.479,E2 -16839.479} C_VEL
LIN {X 0,Y 373.963,Z 589.224,A -85,B 0,C 180,E1 -16841.465,E2 -16841.465} C_VEL
LIN {X 0,Y 372.4,Z 587.865,A -85,B 0,C 180,E1 -16842.326,E2 -16842.326} C_VEL
LIN {X 0,Y 368.367,Z 585.388,A -85,B 0,C 180,E1 -16844.259,E2 -16844.259} C_VEL
LIN {X 0,Y 364.013,Z 581.525,A -85,B 0,C 180,E1 -16846.145,E2 -16846.145} C_VEL
LIN {X 0,Y 361.796,Z 579.593,A -85,B 0,C 180,E1 -16847.024,E2 -16847.024} C_VEL
LIN {X 0,Y 357.294,Z 576.146,A -85,B 0,C 180,E1 -16848.661,E2 -16848.661} C_VEL
LIN {X 0,Y 352.997,Z 572.146,A -85,B 0,C 180,E1 -16850.13,E2 -16850.13} C_VEL
LIN {X 0,Y 348.093,Z 568.041,A -85,B 0,C 180,E1 -16851.671,E2 -16851.671} C_VEL
LIN {X 0,Y 344.404,Z 564.595,A -85,B 0,C 180,E1 -16852.769,E2 -16852.769} C_VEL
LIN {X 0,Y 339.487,Z 560.082,A -85,B 0,C 180,E1 -16854.157,E2 -16854.157} C_VEL
LIN {X 0,Y 335.976,Z 556.796,A -85,B 0,C 180,E1 -16855.103,E2 -16855.103} C_VEL
LIN {X 0,Y 328.353,Z 549.282,A -85,B 0,C 180,E1 -16857.059,E2 -16857.059} C_VEL
LIN {X 0,Y 320.067,Z 540.499,A -85,B 0,C 180,E1 -16859.046,E2 -16859.046} C_VEL
LIN {X 0,Y 314.137,Z 533.933,A -85,B 0,C 180,E1 -16860.343,E2 -16860.343} C_VEL
